// 30 Program Organization Units/FBs/AT_FUNKTIONEN/AT_ANTRIEB_STETIG/FB_AT_ANTRIEB_STETIG
FUNCTION_BLOCK FB_AT_ANTRIEB_STETIG EXTENDS FB_OBJ_ID_BASE
VAR_INPUT
	xRelease		:	BOOL;
	rRelease		:	REAL;
	xSafetyOk		:	BOOL;		
	xHand			:	BOOL;
	xRevision		:	BOOL;
	xAcknowledge	:	BOOL;
	rAcknowledge	:	REAL;
	xCosPhiOk		:	BOOL;
	xErrorAntrieb	:	BOOL;
END_VAR
VAR_OUTPUT
	(* Requests *)
	xHandPrio8	:	BOOL;
END_VAR
VAR
	(* BacNet Objects *)
	A_BO_1				:	WagoSysBACnet.FbBinaryOutput_large(-1);					// Schaltbefehl
	B_TL_1				:	WagoSysBACnet.FbTrendLog_large(-1);                     // Aufzeichnung Betrieb
	C_EE_1				:	WagoSysBACnet.FbEventEnrollment_large(-1);              // Instandhaltungsmeldung
	// Objekt D	wird nicht unterstützt KBOB 2017 AV KBOB 2021 PIV
	E_BV_2				:	WagoSysBACnet.FbBinaryValue_large(-1);                  // Handbetrieb
	F_BI_1				:	WagoSysBACnet.FbBinaryInput_large(-1);                  // Revisionsschalter
	G_AO_1				:	WagoSysBACnet.FbAnalogOutput_large(-1);                 // Sollwertvorgabe
	H_TL_2				:	WagoSysBACnet.FbTrendLog_large(-1);                     // Aufzeichnung Sollwert
	I_AI_1				:	WagoSysBACnet.FbAnalogInput_large(-1);                  // Istwert
	J_TL_3				:	WagoSysBACnet.FbTrendLog_large(-1);                     // Aufzeichnung Istwert
	K_BI_2				:	WagoSysBACnet.FbBinaryInput_large(-1);                  // Lauf Überwachung
	L_BV_3				:	WagoSysBACnet.FbBinaryValue_large(-1);					// Störung Antrieb
END_VAR
VAR CONSTANT
	usiAnzBacNetObj	:	USINT	:= 12;
END_VAR

(* Call Base FB*)
SUPER^();
(* Cyclic Action *)
IF xCreatet THEN
	(* DESCTIPTION FIX *)
	metCYCLIC_DESCRIPTION_FIX();
	(* Get Revision *)
	CASE GVL_BACNET.fbBacNetParameter.proKBOB_REV OF
		(* KBOB 2021 V2 *)
		enKBOB_REV.KBOB_REV2021_V2:
			metCYCLIC_KBOB_2021_V2();
		(* KBOB 2017 V1 *)
		enKBOB_REV.KBOB_REV2017_V1:
			metCYCLIC_KBOB_2017_V1();
		(* Default *)
		ELSE
			metCYCLIC_KBOB_2021_V2();
	END_CASE;	
END_IF;

METHOD metCYCLIC_KBOB_2017_V1
VAR_INPUT
END_VAR
(* A_BO_1 *)
	IF A_BO_1.IPriorityArray.aLevel[16].xValue <> xRelease THEN
		A_BO_1.IPriorityArray.SetPriority(16,xRelease,FALSE);	// Prio 16 Normal Command
	END_IF;
	IF NOT xSafetyOk THEN
		IF A_BO_1.IPriorityArray.aLevel[5].xNull THEN
			A_BO_1.IPriorityArray.SetPriority( 5,FALSE,FALSE);	// Prio  5 Device safety Off
		END_IF;
	ELSE
		IF NOT A_BO_1.IPriorityArray.aLevel[5].xNull THEN
			A_BO_1.IPriorityArray.SetPriority( 5,FALSE,TRUE);	// Prio  5 Device safety NULL
		END_IF;
	END_IF;	
	IF A_BO_1.xFeedbackValue <> xAcknowledge THEN
		A_BO_1.xFeedbackValue := xAcknowledge;
	END_IF;

	(* E_BV_2 *)
	IF E_BV_2.IPriorityArray.aLevel[16].xValue <> (xHand OR xRevision) THEN
		E_BV_2.IPriorityArray.SetPriority(16,xHand OR xRevision,FALSE);
	END_IF;
	(* F_BI_1 *)
	F_BI_1.xIN := xRevision;
	(* G_AO_1 *)
	IF G_AO_1.IPriorityArray.aLevel[5].rValue <> rRelease THEN
		G_AO_1.IPriorityArray.SetPriority(5,rRelease,FALSE);
	END_IF;
	(* I_AI_1 *)
	I_AI_1.rIN := rAcknowledge;
	(* K_BI_2 *)
	K_BI_2.xIN := xCosPhiOk;
	(* L_BV_3 *)
	L_BV_3.xPresentValue := xErrorAntrieb;
	
	(* Request Hand Prio 8 *)
	xHandPrio8 := NOT A_BO_1.IPriorityArray.aLevel[8].xNull AND A_BO_1.IPriorityArray.aLevel[8].xValue;
END_METHOD

METHOD metCYCLIC_KBOB_2021_V2
VAR_INPUT
END_VAR
(* A_BO_1 *)
	IF A_BO_1.IPriorityArray.aLevel[16].xValue <> xRelease THEN
		A_BO_1.IPriorityArray.SetPriority(16,xRelease,FALSE);	// Prio 16 Normal Command
	END_IF;
	IF NOT xSafetyOk THEN
		IF A_BO_1.IPriorityArray.aLevel[5].xNull THEN
			A_BO_1.IPriorityArray.SetPriority( 5,FALSE,FALSE);	// Prio  5 Device safety Off
		END_IF;
	ELSE
		IF NOT A_BO_1.IPriorityArray.aLevel[5].xNull THEN
			A_BO_1.IPriorityArray.SetPriority( 5,FALSE,TRUE);	// Prio  5 Device safety NULL
		END_IF;
	END_IF;	
	IF A_BO_1.xFeedbackValue <> xAcknowledge THEN
		A_BO_1.xFeedbackValue := xAcknowledge;
	END_IF;

	(* E_BV_2 *)
	IF E_BV_2.IPriorityArray.aLevel[16].xValue <> (xHand OR xRevision) THEN
		E_BV_2.IPriorityArray.SetPriority(16,xHand OR xRevision,FALSE);
	END_IF;
	(* F_BI_1 *)
	F_BI_1.xIN := xRevision;
	(* G_AO_1 *)
	IF G_AO_1.IPriorityArray.aLevel[5].rValue <> rRelease THEN
		G_AO_1.IPriorityArray.SetPriority(5,rRelease,FALSE);
	END_IF;
	(* I_AI_1 *)
	I_AI_1.rIN := rAcknowledge;
	(* K_BI_2 *)
	K_BI_2.xIN := xCosPhiOk;
	(* L_BV_3 *)
	L_BV_3.xPresentValue := xErrorAntrieb;
	
	(* Request Hand Prio 8 *)
	xHandPrio8 := NOT A_BO_1.IPriorityArray.aLevel[8].xNull AND A_BO_1.IPriorityArray.aLevel[8].xValue;
END_METHOD

METHOD metCYCLIC_DESCRIPTION_FIX
VAR_INPUT
END_VAR
(* A_BO_1 *)
IF A_BO_1.xIsCreated THEN
	IF A_BO_1.sDescription <> A_BO_1._sDescription THEN
		A_BO_1.sDescription := A_BO_1._sDescription;
	END_IF;
END_IF;

(* B_TL_1 *)
IF B_TL_1.xIsCreated THEN
	IF B_TL_1.sDescription <> B_TL_1._sDescription THEN
		B_TL_1.sDescription := B_TL_1._sDescription;
	END_IF;
END_IF;

(* C_EE_1 *)
IF C_EE_1.xIsCreated THEN
	IF C_EE_1.sDescription <> C_EE_1._sDescription THEN
		C_EE_1.sDescription := C_EE_1._sDescription;
	END_IF;
END_IF;

(* D_ *)
// Not Avaiable

(* E_BV_2 *)
IF E_BV_2.xIsCreated THEN
	IF E_BV_2.sDescription <> E_BV_2._sDescription THEN
		E_BV_2.sDescription := E_BV_2._sDescription;
	END_IF;
END_IF;

(* F_BI_1 *)
IF F_BI_1.xIsCreated THEN
	IF F_BI_1.sDescription <> F_BI_1._sDescription THEN
		F_BI_1.sDescription := F_BI_1._sDescription;
	END_IF;
END_IF;

(* G_AO_1 *)
IF G_AO_1.xIsCreated THEN
	IF G_AO_1.sDescription <> G_AO_1._sDescription THEN
		G_AO_1.sDescription := G_AO_1._sDescription;
	END_IF;
END_IF;

(* H_TL_2 *)
IF H_TL_2.xIsCreated THEN
	IF H_TL_2.sDescription <> H_TL_2._sDescription THEN
		H_TL_2.sDescription := H_TL_2._sDescription;
	END_IF;
END_IF;

(* I_AI_1 *)
IF I_AI_1.xIsCreated THEN
	IF I_AI_1.sDescription <> I_AI_1._sDescription THEN
		I_AI_1.sDescription := I_AI_1._sDescription;
	END_IF;
END_IF;

(* J_TL_3 *)
IF J_TL_3.xIsCreated THEN
	IF J_TL_3.sDescription <> J_TL_3._sDescription THEN
		J_TL_3.sDescription := J_TL_3._sDescription;
	END_IF;
END_IF;

(* K_BI_2 *)
IF K_BI_2.xIsCreated THEN
	IF K_BI_2.sDescription <> K_BI_2._sDescription THEN
		K_BI_2.sDescription := K_BI_2._sDescription;
	END_IF;
END_IF;

(* L_BV_3 *)
IF L_BV_3.xIsCreated THEN
	IF L_BV_3.sDescription <> L_BV_3._sDescription THEN
		L_BV_3.sDescription := L_BV_3._sDescription;
	END_IF;
END_IF;
END_METHOD

(*FB_Exit muss explizit implementiert werden. Wenn es eine Implementierung gibt, dann wird 
die Methode aufgerufen, bevor die Steuerung den Code der Funktionsbaustein-Instanz entfernt
(impliziter Aufruf. Der Rückgabewert wird nicht ausgewertet.*)
METHOD FB_Exit : BOOL
VAR_INPUT
	(* TRUE: Die Exit-Methode wird aufgerufen, um die Instanz zu verlassen, die hinterher kopiert wird Online-Change).  *)
	bInCopyCode	: BOOL;
END_VAR
(* A_BO_1*)
IF A_BO_1.xIsCreated THEN
	A_BO_1.Delete();
END_IF;	
(* B_TL_1 *)
IF B_TL_1.xIsCreated THEN
	B_TL_1.Delete();
END_IF;	
(* C_EE_1 *)
IF C_EE_1.xIsCreated THEN
	C_EE_1.Delete();
END_IF;
(* E_BV_2 *)
IF E_BV_2.xIsCreated THEN
	E_BV_2.Delete();
END_IF;
(* F_BI_1 *)
IF F_BI_1.xIsCreated THEN
	F_BI_1.Delete();	
END_IF;
(* G_AO_1 *)
IF G_AO_1.xIsCreated THEN
	G_AO_1.Delete();
END_IF;
(* H_TL_2 *)
IF H_TL_2.xIsCreated THEN
	H_TL_2.Delete();
END_IF;
(* I_AI_1 *)
IF I_AI_1.xIsCreated THEN
	I_AI_1.Delete();
END_IF;
(* J_TL_3 *)
IF J_TL_3.xIsCreated THEN
	J_TL_3.Delete();
END_IF;
(* K_BI_2 *)
IF K_BI_2.xIsCreated THEN
	K_BI_2.Delete();
END_IF;
(* L_BV_3 *)
IF L_BV_3.xIsCreated THEN
	L_BV_3.Delete();
END_IF;
END_METHOD

METHOD metDELETE : BOOL
VAR_INPUT
END_VAR
VAR
	oStatus		:	WagoSysErrorBase.FbResult;
END_VAR
(* A_BO_1*)
IF A_BO_1.xIsCreated THEN
	A_BO_1.Delete(oStatus=>oStatus);
END_IF;	
(* B_TL_1 *)
IF B_TL_1.xIsCreated THEN
	IF GVL_BACNET.fbBacNetParameter.proDestroyBacNetOverrideXmlNode THEN
		fcXMLDeleteOverrideNode(fcBacNetIdToIdWitType(B_TL_1.IObjectIdentifier.diInstance,B_TL_1.IObjectIdentifier.eObjectType));
	END_IF;
	B_TL_1.Delete(oStatus=>oStatus);
END_IF;	
(* C_EE_1 *)
IF C_EE_1.xIsCreated THEN
	C_EE_1.Delete(oStatus=>oStatus);
END_IF;
(* E_BV_2 *)
IF E_BV_2.xIsCreated THEN
	E_BV_2.Delete(oStatus=>oStatus);
END_IF;
(* F_BI_1 *)
IF F_BI_1.xIsCreated THEN
	F_BI_1.Delete(oStatus=>oStatus);	
END_IF;
(* G_AO_1 *)
IF G_AO_1.xIsCreated THEN
	G_AO_1.Delete(oStatus=>oStatus);
END_IF;
(* H_TL_2 *)
IF H_TL_2.xIsCreated THEN
	IF GVL_BACNET.fbBacNetParameter.proDestroyBacNetOverrideXmlNode THEN
		fcXMLDeleteOverrideNode(fcBacNetIdToIdWitType(H_TL_2.IObjectIdentifier.diInstance,H_TL_2.IObjectIdentifier.eObjectType));
	END_IF;
	H_TL_2.Delete(oStatus=>oStatus);
END_IF;
(* I_AI_1 *)
IF I_AI_1.xIsCreated THEN
	I_AI_1.Delete(oStatus=>oStatus);
END_IF;
(* J_TL_3 *)
IF J_TL_3.xIsCreated THEN
	IF GVL_BACNET.fbBacNetParameter.proDestroyBacNetOverrideXmlNode THEN
		fcXMLDeleteOverrideNode(fcBacNetIdToIdWitType(J_TL_3.IObjectIdentifier.diInstance,J_TL_3.IObjectIdentifier.eObjectType));
	END_IF;
	J_TL_3.Delete(oStatus=>oStatus);
END_IF;
(* K_BI_2 *)
IF K_BI_2.xIsCreated THEN
	K_BI_2.Delete(oStatus=>oStatus);
END_IF;
(* L_BV_3 *)
IF L_BV_3.xIsCreated THEN
	L_BV_3.Delete(oStatus=>oStatus);
END_IF;
(* Delete Struct View *)
IF GVL_BACNET.fbBacNetParameter.proDestroyBacNetOverrideXmlNode THEN
	fcXMLDeleteOverrideNode(fcBacNetIdToIdWitType(TO_DINT(CONCAT(TO_STRING(OBJ_ID_BASE),'1')),WagoTypesBacNet.eBACnetObjectType.BACnet_structured_view));
	fcXMLDeleteStructuredViewFromDevice(fcBacNetIdToIdWitType(TO_DINT(CONCAT(TO_STRING(OBJ_ID_BASE),'1')),WagoTypesBacNet.eBACnetObjectType.BACnet_structured_view));
END_IF;
metDELETE := 	A_BO_1.xIsCreated OR 
				B_TL_1.xIsCreated OR
				C_EE_1.xIsCreated OR				
				E_BV_2.xIsCreated OR
				F_BI_1.xIsCreated OR
				G_AO_1.xIsCreated OR
				I_AI_1.xIsCreated OR
				K_BI_2.xIsCreated OR
				L_BV_3.xIsCreated;
(* Reset Create Case *)
usiCreateCase := 1;
END_METHOD

METHOD metCREATE_KBOB_2017_V1 : BOOL;
VAR_INPUT
END_VAR
VAR
	oStatus		:	WagoSysErrorBase.FbResult;
	usiErrors	:	USINT;
END_VAR
(* Resett *)
usiErrors := 0;	

(* Create Objeccts *)
CASE usiCreateCase OF
	1:	
		usiErrors := usiErrors + TO_USINT(NOT metCreate_A_BO_1());
	2:
		usiErrors := usiErrors + TO_USINT(NOT metCreate_B_TL_1());
	3:	
		usiErrors := usiErrors + TO_USINT(NOT metCreate_C_EE_1());
	4:	
		;// Objekt D aus KBOB 2017 nicht realisierbar aufgrund fehlender Setpoint reference
	5:
		usiErrors := usiErrors + TO_USINT(NOT metCreate_E_BV_2());
	6:	
		usiErrors := usiErrors + TO_USINT(NOT metCreate_F_BI_1());
	7:
		usiErrors := usiErrors + TO_USINT(NOT metCreate_G_AO_1());
	8:	
		usiErrors := usiErrors + TO_USINT(NOT metCreate_H_TL_2());
	9:
		usiErrors := usiErrors + TO_USINT(NOT metCreate_I_AI_1());
	10:
		usiErrors := usiErrors + TO_USINT(NOT metCreate_J_TL_3());
	11:	
		usiErrors := usiErrors + TO_USINT(NOT metCreate_K_BI_2());
	12:
		usiErrors := usiErrors + TO_USINT(NOT metCreate_L_BV_3());
	0: 
		usiCreateCase := 1;
ELSE
	usiCreateCase := 0;
END_CASE;

(* STRUCT VIEW *)
metCREATE_STRUCTVIEW_KBOB_2017_V1();

(* OK = 0*)
metCREATE_KBOB_2017_V1 := NOT TO_BOOL(usiErrors);
END_METHOD

METHOD metCREATE_STRUCTVIEW_KBOB_2017_V1 : BOOL
VAR_INPUT
END_VAR
CASE usiCreateCase OF
	1:
		fcXMLStructuredView(THIS^,A_BO_1.IObjectIdentifier);
	2:
		fcXMLStructuredView(THIS^,B_TL_1.IObjectIdentifier);
	3:
		fcXMLStructuredView(THIS^,C_EE_1.IObjectIdentifier);
	4:
		;// Reserve für D
	5:
		fcXMLStructuredView(THIS^,E_BV_2.IObjectIdentifier);
	6:
		fcXMLStructuredView(THIS^,F_BI_1.IObjectIdentifier);
	7:
		fcXMLStructuredView(THIS^,G_AO_1.IObjectIdentifier);
	8:
		fcXMLStructuredView(THIS^,H_TL_2.IObjectIdentifier);
	9:
		fcXMLStructuredView(THIS^,I_AI_1.IObjectIdentifier);
	10:
		fcXMLStructuredView(THIS^,J_TL_3.IObjectIdentifier);
	11:
		fcXMLStructuredView(THIS^,K_BI_2.IObjectIdentifier);
	12:
		fcXMLStructuredView(THIS^,L_BV_3.IObjectIdentifier);
		fcXMLAddStructuredViewToDevice(THIS^);	
	0: 
		usiCreateCase := 1;
ELSE
	usiCreateCase := 0;
END_CASE
END_METHOD

METHOD metCREATE_STRUCTVIEW_KBOB_2021_V2 : BOOL
VAR_INPUT
END_VAR
CASE usiCreateCase OF
	1:
		fcXMLStructuredView(THIS^,A_BO_1.IObjectIdentifier);
	2:
		fcXMLStructuredView(THIS^,B_TL_1.IObjectIdentifier);
	3:
		fcXMLStructuredView(THIS^,C_EE_1.IObjectIdentifier);
	4:
		;// Reserve für D
	5:
		fcXMLStructuredView(THIS^,E_BV_2.IObjectIdentifier);
	6:
		fcXMLStructuredView(THIS^,F_BI_1.IObjectIdentifier);
	7:
		fcXMLStructuredView(THIS^,G_AO_1.IObjectIdentifier);
	8:
		fcXMLStructuredView(THIS^,H_TL_2.IObjectIdentifier);
	9:
		fcXMLStructuredView(THIS^,I_AI_1.IObjectIdentifier);
	10:
		fcXMLStructuredView(THIS^,J_TL_3.IObjectIdentifier);
	11:
		fcXMLStructuredView(THIS^,K_BI_2.IObjectIdentifier);
	12:
		fcXMLStructuredView(THIS^,L_BV_3.IObjectIdentifier);
		fcXMLAddStructuredViewToDevice(THIS^);	
	0: 
		usiCreateCase := 1;
ELSE
	usiCreateCase := 0;
END_CASE
END_METHOD

METHOD metCREATE_KBOB_2021_V2 : BOOL;
VAR_INPUT
END_VAR
VAR
	oStatus		:	WagoSysErrorBase.FbResult;
	usiErrors	:	USINT;
END_VAR
(* Resett *)
usiErrors := 0;	

(* Create Objeccts *)
CASE usiCreateCase OF
	1:	
		usiErrors := usiErrors + TO_USINT(NOT metCreate_A_BO_1());
	2:
		usiErrors := usiErrors + TO_USINT(NOT metCreate_B_TL_1());
	3:	
		usiErrors := usiErrors + TO_USINT(NOT metCreate_C_EE_1());
	4:	
		;// Objekt D aus KBOB 2017 nicht realisierbar aufgrund fehlender Setpoint reference
	5:
		usiErrors := usiErrors + TO_USINT(NOT metCreate_E_BV_2());
	6:	
		usiErrors := usiErrors + TO_USINT(NOT metCreate_F_BI_1());
	7:
		usiErrors := usiErrors + TO_USINT(NOT metCreate_G_AO_1());
	8:	
		usiErrors := usiErrors + TO_USINT(NOT metCreate_H_TL_2());
	9:
		usiErrors := usiErrors + TO_USINT(NOT metCreate_I_AI_1());
	10:
		usiErrors := usiErrors + TO_USINT(NOT metCreate_J_TL_3());
	11:	
		usiErrors := usiErrors + TO_USINT(NOT metCreate_K_BI_2());
	12:
		usiErrors := usiErrors + TO_USINT(NOT metCreate_L_BV_3());
	0: 
		usiCreateCase := 1;
ELSE
	usiCreateCase := 0;
END_CASE;

(* STRUCT VIEW *)
metCREATE_STRUCTVIEW_KBOB_2021_V2();

(* OK = 0*)
metCREATE_KBOB_2021_V2 := NOT TO_BOOL(usiErrors);
END_METHOD

METHOD metCREATE : BOOL;
VAR_INPUT
END_VAR
VAR
	oStatus		:	WagoSysErrorBase.FbResult;
	usiErrors	:	USINT;
END_VAR
(* Get Revision *)
CASE GVL_BACNET.fbBacNetParameter.proKBOB_REV OF
	(* KBOB 2021 V2 *)
	enKBOB_REV.KBOB_REV2021_V2:
		usiErrors := usiErrors + TO_USINT(NOT metCREATE_KBOB_2021_V2());
	(* KBOB 2017 V1 *)
	enKBOB_REV.KBOB_REV2017_V1:
		usiErrors := usiErrors + TO_USINT(NOT metCREATE_KBOB_2017_V1());
	(* Default *)
	ELSE
		usiErrors := usiErrors + TO_USINT(NOT metCREATE_KBOB_2021_V2());
END_CASE;

(* OK = 0*)
xErrorCreate := TO_BOOL(usiErrors);
metCREATE := NOT TO_BOOL(usiErrors) AND usiCreateCase = usiAnzBacNetObj;
END_METHOD

METHOD metCreate_F_BI_1 : BOOL
(* F_BI_1*)
IF NOT F_BI_1.xIsCreated THEN
	(* Ziel						UTF8->ASCII						OBJ_NAME_BASE			BacNet Text		Textlistname									BacNet Funktion																BacNet Textlist type												TextId		*)
	F_BI_1._sObjectName		:=	fcUtfToAscii(Standard.CONCAT(	OBJ_NAME_BASE		,	fcGetBcText(	GVL_BACNET.fbBacNetParameter.metGetTextListName(enTypeOfBacNetFunktionIn := enTypeOfBacNetFunktion.Type_AntriebStetig,		enTypeOfBacNetTextListIn := enTypeOfBacNetTextList.ENDING		),	'F_BI_1')));
	F_BI_1._sDescription	:= 	fcUtfToAscii(Standard.CONCAT(	OBJ_NAME_DESCRIPTION,	fcGetBcText(	GVL_BACNET.fbBacNetParameter.metGetTextListName(enTypeOfBacNetFunktionIn := enTypeOfBacNetFunktion.Type_AntriebStetig,		enTypeOfBacNetTextListIn := enTypeOfBacNetTextList.DESCRIPTION	),	'F_BI_1')));
	(* Create Id from Base Id and Object Nr (Last nummber of Name *)	
	F_BI_1.Create(diInstance := TO_DINT(Standard.CONCAT(TO_STRING(dwOBJ_ID_BASE),'1')));
	(* Check if Created *)
	IF F_BI_1.xIsCreated THEN
		(* Set Group *)
		F_BI_1.setPropertyGroup(WagoTypesBacNet.eBACnetPropertyIdentifier.PROP_PRESENT_VALUE						,WagoTypesBacNet.eBACnetPropertyUpdateGroup.GROUP_CYCLIC);
		F_BI_1.setPropertyGroup(WagoTypesBacNet.eBACnetPropertyIdentifier.PROP_PRIORITY_ARRAY						,WagoTypesBacNet.eBACnetPropertyUpdateGroup.GROUP_CYCLIC);
		F_BI_1.setPropertyGroup(WagoTypesBacNet.eBACnetPropertyIdentifier.PROP_ELAPSED_ACTIVE_TIME					,WagoTypesBacNet.eBACnetPropertyUpdateGroup.GROUP_CYCLIC);
		F_BI_1.setPropertyGroup(WagoTypesBacNet.eBACnetPropertyIdentifier.PROP_DESCRIPTION							,WagoTypesBacNet.eBACnetPropertyUpdateGroup.GROUP_CYCLIC);
		F_BI_1.setPropertyGroup(WagoTypesBacNet.eBACnetPropertyIdentifier.PROP_EVENT_MESSAGE_TEXTS_CONFIG			,WagoTypesBacNet.eBACnetPropertyUpdateGroup.GROUP_CYCLIC);
				
		(* Ziel												UTF8->ASCII		BacNet Text		Textlistname									BacNet Funktion																BacNet Textlist type												TextId		*)
		F_BI_1.IEventMessageTextsConfig.sToOffNormal	:=	fcUtfToAscii(	fcGetBcText(	GVL_BACNET.fbBacNetParameter.metGetTextListName(enTypeOfBacNetFunktionIn := enTypeOfBacNetFunktion.Type_AntriebStetig,		enTypeOfBacNetTextListIn := enTypeOfBacNetTextList.EVENTMESSAGE	),	'F_BI_1_ToOffNormal'	));		
		F_BI_1.IEventMessageTextsConfig.sToFault		:=	fcUtfToAscii(	fcGetBcText(	GVL_BACNET.fbBacNetParameter.metGetTextListName(enTypeOfBacNetFunktionIn := enTypeOfBacNetFunktion.Type_AntriebStetig,		enTypeOfBacNetTextListIn := enTypeOfBacNetTextList.EVENTMESSAGE	),	'F_BI_1_ToFault'		));		
		F_BI_1.IEventMessageTextsConfig.sToNormal		:=	fcUtfToAscii(	fcGetBcText(	GVL_BACNET.fbBacNetParameter.metGetTextListName(enTypeOfBacNetFunktionIn := enTypeOfBacNetFunktion.Type_AntriebStetig,		enTypeOfBacNetTextListIn := enTypeOfBacNetTextList.EVENTMESSAGE	),	'F_BI_1_ToNormal'		));		

		(* Ziel												UTF8->ASCII		BacNet Text		Textlistname									BacNet Funktion																BacNet Textlist type												TextId		*)	
		F_BI_1.sActiveText								:= 	fcUtfToAscii(	fcGetBcText(	GVL_BACNET.fbBacNetParameter.metGetTextListName(enTypeOfBacNetFunktionIn := enTypeOfBacNetFunktion.Type_AntriebStetig,		enTypeOfBacNetTextListIn := enTypeOfBacNetTextList.PRESENTVALUE	),	'F_BI_1_ST_ACTIVE'		));
		F_BI_1.sInactiveText							:= 	fcUtfToAscii(	fcGetBcText(	GVL_BACNET.fbBacNetParameter.metGetTextListName(enTypeOfBacNetFunktionIn := enTypeOfBacNetFunktion.Type_AntriebStetig,		enTypeOfBacNetTextListIn := enTypeOfBacNetTextList.PRESENTVALUE	),	'F_BI_1_ST_INACTIVE'	));	

		(* Ziel												Convert			BacNet Text		Textlistname									BacNet Funktion																BacNet Textlist type												TextId		*)	
		F_BI_1.udiNotificationClass						:= 	TO_UDINT	(	fcGetBcText(	GVL_BACNET.fbBacNetParameter.metGetTextListName(enTypeOfBacNetFunktionIn := enTypeOfBacNetFunktion.Type_AntriebStetig,		enTypeOfBacNetTextListIn := enTypeOfBacNetTextList.NC			),	'F_BI_1_NC'	));	
		F_BI_1.eNotifyType								:= 	WagoTypesBACnet.eBACnetNotifyType.NOTIFY_TYPE_EVENT;
		F_BI_1.xAlarmValue								:= 	TO_BOOL		(	fcGetBcText(	GVL_BACNET.fbBacNetParameter.metGetTextListName(enTypeOfBacNetFunktionIn := enTypeOfBacNetFunktion.Type_AntriebStetig,		enTypeOfBacNetTextListIn := enTypeOfBacNetTextList.NC			),	'F_BI_1_ALV'	));	
		
	ELSE
		F_BI_1.Delete();
	END_IF;
	(* Get Status *)
	metCreate_F_BI_1 := F_BI_1.xIsCreated;	
END_IF;
END_METHOD

METHOD metCreate_G_AO_1 : BOOL
(* G_AO_1*)
IF NOT G_AO_1.xIsCreated THEN
	(* Ziel						UTF8->ASCII						OBJ_NAME_BASE			BacNet Text		Textlistname									BacNet Funktion																BacNet Textlist type												TextId		*)
	G_AO_1._sObjectName		:=	fcUtfToAscii(Standard.CONCAT(	OBJ_NAME_BASE		,	fcGetBcText(	GVL_BACNET.fbBacNetParameter.metGetTextListName(enTypeOfBacNetFunktionIn := enTypeOfBacNetFunktion.Type_AntriebStetig,		enTypeOfBacNetTextListIn := enTypeOfBacNetTextList.ENDING		),	'G_AO_1')));
	G_AO_1._sDescription	:= 	fcUtfToAscii(Standard.CONCAT(	OBJ_NAME_DESCRIPTION,	fcGetBcText(	GVL_BACNET.fbBacNetParameter.metGetTextListName(enTypeOfBacNetFunktionIn := enTypeOfBacNetFunktion.Type_AntriebStetig,		enTypeOfBacNetTextListIn := enTypeOfBacNetTextList.DESCRIPTION	),	'G_AO_1')));
	(* Create Id from Base Id and Object Nr (Last nummber of Name *)	
	G_AO_1.Create(diInstance := TO_DINT(Standard.CONCAT(TO_STRING(dwOBJ_ID_BASE),'1')));
	(* Check if Created *)
	IF G_AO_1.xIsCreated THEN
		(* Set Group *)
		G_AO_1.setPropertyGroup(WagoTypesBacNet.eBACnetPropertyIdentifier.PROP_PRESENT_VALUE						,WagoTypesBacNet.eBACnetPropertyUpdateGroup.GROUP_CYCLIC);
		G_AO_1.setPropertyGroup(WagoTypesBacNet.eBACnetPropertyIdentifier.PROP_PRIORITY_ARRAY						,WagoTypesBacNet.eBACnetPropertyUpdateGroup.GROUP_CYCLIC);
		G_AO_1.setPropertyGroup(WagoTypesBacNet.eBACnetPropertyIdentifier.PROP_ELAPSED_ACTIVE_TIME					,WagoTypesBacNet.eBACnetPropertyUpdateGroup.GROUP_CYCLIC);
		G_AO_1.setPropertyGroup(WagoTypesBacNet.eBACnetPropertyIdentifier.PROP_DESCRIPTION							,WagoTypesBacNet.eBACnetPropertyUpdateGroup.GROUP_CYCLIC);
		G_AO_1.setPropertyGroup(WagoTypesBacNet.eBACnetPropertyIdentifier.PROP_EVENT_MESSAGE_TEXTS_CONFIG			,WagoTypesBacNet.eBACnetPropertyUpdateGroup.GROUP_CYCLIC);
				
		(* Ziel												UTF8->ASCII		BacNet Text		Textlistname									BacNet Funktion																BacNet Textlist type												TextId		*)
		G_AO_1.IEventMessageTextsConfig.sToOffNormal	:=	fcUtfToAscii(	fcGetBcText(	GVL_BACNET.fbBacNetParameter.metGetTextListName(enTypeOfBacNetFunktionIn := enTypeOfBacNetFunktion.Type_AntriebStetig,		enTypeOfBacNetTextListIn := enTypeOfBacNetTextList.EVENTMESSAGE	),	'G_AO_1_ToOffNormal'	));		
		G_AO_1.IEventMessageTextsConfig.sToFault		:=	fcUtfToAscii(	fcGetBcText(	GVL_BACNET.fbBacNetParameter.metGetTextListName(enTypeOfBacNetFunktionIn := enTypeOfBacNetFunktion.Type_AntriebStetig,		enTypeOfBacNetTextListIn := enTypeOfBacNetTextList.EVENTMESSAGE	),	'G_AO_1_ToFault'		));		
		G_AO_1.IEventMessageTextsConfig.sToNormal		:=	fcUtfToAscii(	fcGetBcText(	GVL_BACNET.fbBacNetParameter.metGetTextListName(enTypeOfBacNetFunktionIn := enTypeOfBacNetFunktion.Type_AntriebStetig,		enTypeOfBacNetTextListIn := enTypeOfBacNetTextList.EVENTMESSAGE	),	'G_AO_1_ToNormal'		));		

	ELSE
		G_AO_1.Delete();
	END_IF;
	(* Get Status *)
	metCreate_G_AO_1 := G_AO_1.xIsCreated;	
END_IF;
END_METHOD

METHOD metCreate_I_AI_1 : BOOL
(* I_AI_1*)
IF NOT I_AI_1.xIsCreated THEN
	(* Ziel						UTF8->ASCII						OBJ_NAME_BASE			BacNet Text		Textlistname									BacNet Funktion																BacNet Textlist type												TextId		*)
	I_AI_1._sObjectName		:=	fcUtfToAscii(Standard.CONCAT(	OBJ_NAME_BASE		,	fcGetBcText(	GVL_BACNET.fbBacNetParameter.metGetTextListName(enTypeOfBacNetFunktionIn := enTypeOfBacNetFunktion.Type_AntriebStetig,		enTypeOfBacNetTextListIn := enTypeOfBacNetTextList.ENDING		),	'I_AI_1')));
	I_AI_1._sDescription	:= 	fcUtfToAscii(Standard.CONCAT(	OBJ_NAME_DESCRIPTION,	fcGetBcText(	GVL_BACNET.fbBacNetParameter.metGetTextListName(enTypeOfBacNetFunktionIn := enTypeOfBacNetFunktion.Type_AntriebStetig,		enTypeOfBacNetTextListIn := enTypeOfBacNetTextList.DESCRIPTION	),	'I_AI_1')));
	(* Create Id from Base Id and Object Nr (Last nummber of Name *)	
	I_AI_1.Create(diInstance := TO_DINT(Standard.CONCAT(TO_STRING(dwOBJ_ID_BASE),'1')));
	(* Check if Created *)
	IF I_AI_1.xIsCreated THEN
		(* Set Group *)
		I_AI_1.setPropertyGroup(WagoTypesBacNet.eBACnetPropertyIdentifier.PROP_PRESENT_VALUE						,WagoTypesBacNet.eBACnetPropertyUpdateGroup.GROUP_CYCLIC);
		I_AI_1.setPropertyGroup(WagoTypesBacNet.eBACnetPropertyIdentifier.PROP_PRIORITY_ARRAY						,WagoTypesBacNet.eBACnetPropertyUpdateGroup.GROUP_CYCLIC);
		I_AI_1.setPropertyGroup(WagoTypesBacNet.eBACnetPropertyIdentifier.PROP_ELAPSED_ACTIVE_TIME					,WagoTypesBacNet.eBACnetPropertyUpdateGroup.GROUP_CYCLIC);
		I_AI_1.setPropertyGroup(WagoTypesBacNet.eBACnetPropertyIdentifier.PROP_DESCRIPTION							,WagoTypesBacNet.eBACnetPropertyUpdateGroup.GROUP_CYCLIC);
		I_AI_1.setPropertyGroup(WagoTypesBacNet.eBACnetPropertyIdentifier.PROP_EVENT_MESSAGE_TEXTS_CONFIG			,WagoTypesBacNet.eBACnetPropertyUpdateGroup.GROUP_CYCLIC);
		
		(* Ziel												UTF8->ASCII		BacNet Text		Textlistname									BacNet Funktion																BacNet Textlist type												TextId		*)
		I_AI_1.IEventMessageTextsConfig.sToOffNormal	:=	fcUtfToAscii(	fcGetBcText(	GVL_BACNET.fbBacNetParameter.metGetTextListName(enTypeOfBacNetFunktionIn := enTypeOfBacNetFunktion.Type_AntriebStetig,		enTypeOfBacNetTextListIn := enTypeOfBacNetTextList.EVENTMESSAGE	),	'I_AI_1_ToOffNormal'	));		
		I_AI_1.IEventMessageTextsConfig.sToFault		:=	fcUtfToAscii(	fcGetBcText(	GVL_BACNET.fbBacNetParameter.metGetTextListName(enTypeOfBacNetFunktionIn := enTypeOfBacNetFunktion.Type_AntriebStetig,		enTypeOfBacNetTextListIn := enTypeOfBacNetTextList.EVENTMESSAGE	),	'I_AI_1_ToFault'		));		
		I_AI_1.IEventMessageTextsConfig.sToNormal		:=	fcUtfToAscii(	fcGetBcText(	GVL_BACNET.fbBacNetParameter.metGetTextListName(enTypeOfBacNetFunktionIn := enTypeOfBacNetFunktion.Type_AntriebStetig,		enTypeOfBacNetTextListIn := enTypeOfBacNetTextList.EVENTMESSAGE	),	'I_AI_1_ToNormal'		));		

		(* Ziel												Convert			BacNet Text		Textlistname									BacNet Funktion																BacNet Textlist type												TextId		*)	
		I_AI_1.udiNotificationClass						:= 	TO_UDINT	(	fcGetBcText(	GVL_BACNET.fbBacNetParameter.metGetTextListName(enTypeOfBacNetFunktionIn := enTypeOfBacNetFunktion.Type_AntriebStetig,		enTypeOfBacNetTextListIn := enTypeOfBacNetTextList.NC			),	'I_AI_1_NC'	));	
		I_AI_1.eNotifyType								:= 	WagoTypesBACnet.eBACnetNotifyType.NOTIFY_TYPE_EVENT;
		
	ELSE
		I_AI_1.Delete();
	END_IF;
	(* Get Status *)
	metCreate_I_AI_1 := I_AI_1.xIsCreated;	
END_IF;
END_METHOD

METHOD metCreate_K_BI_2 : BOOL
(* K_BI_2*)
IF NOT K_BI_2.xIsCreated THEN
	(* Ziel						UTF8->ASCII						OBJ_NAME_BASE			BacNet Text		Textlistname									BacNet Funktion																BacNet Textlist type												TextId		*)
	K_BI_2._sObjectName		:=	fcUtfToAscii(Standard.CONCAT(	OBJ_NAME_BASE		,	fcGetBcText(	GVL_BACNET.fbBacNetParameter.metGetTextListName(enTypeOfBacNetFunktionIn := enTypeOfBacNetFunktion.Type_AntriebStetig,		enTypeOfBacNetTextListIn := enTypeOfBacNetTextList.ENDING		),	'K_BI_2')));
	K_BI_2._sDescription	:= 	fcUtfToAscii(Standard.CONCAT(	OBJ_NAME_DESCRIPTION,	fcGetBcText(	GVL_BACNET.fbBacNetParameter.metGetTextListName(enTypeOfBacNetFunktionIn := enTypeOfBacNetFunktion.Type_AntriebStetig,		enTypeOfBacNetTextListIn := enTypeOfBacNetTextList.DESCRIPTION	),	'K_BI_2')));
	(* Create Id from Base Id and Object Nr (Last nummber of Name *)	
	K_BI_2.Create(diInstance := TO_DINT(Standard.CONCAT(TO_STRING(dwOBJ_ID_BASE),'2')));
	(* Check if Created *)
	IF K_BI_2.xIsCreated THEN
		(* Set Group *)
		K_BI_2.setPropertyGroup(WagoTypesBacNet.eBACnetPropertyIdentifier.PROP_PRESENT_VALUE						,WagoTypesBacNet.eBACnetPropertyUpdateGroup.GROUP_CYCLIC);
		K_BI_2.setPropertyGroup(WagoTypesBacNet.eBACnetPropertyIdentifier.PROP_PRIORITY_ARRAY						,WagoTypesBacNet.eBACnetPropertyUpdateGroup.GROUP_CYCLIC);
		K_BI_2.setPropertyGroup(WagoTypesBacNet.eBACnetPropertyIdentifier.PROP_ELAPSED_ACTIVE_TIME					,WagoTypesBacNet.eBACnetPropertyUpdateGroup.GROUP_CYCLIC);
		K_BI_2.setPropertyGroup(WagoTypesBacNet.eBACnetPropertyIdentifier.PROP_DESCRIPTION							,WagoTypesBacNet.eBACnetPropertyUpdateGroup.GROUP_CYCLIC);
		K_BI_2.setPropertyGroup(WagoTypesBacNet.eBACnetPropertyIdentifier.PROP_EVENT_MESSAGE_TEXTS_CONFIG			,WagoTypesBacNet.eBACnetPropertyUpdateGroup.GROUP_CYCLIC);
		
		(* Ziel												UTF8->ASCII		BacNet Text		Textlistname									BacNet Funktion																BacNet Textlist type												TextId		*)
		K_BI_2.IEventMessageTextsConfig.sToOffNormal	:=	fcUtfToAscii(	fcGetBcText(	GVL_BACNET.fbBacNetParameter.metGetTextListName(enTypeOfBacNetFunktionIn := enTypeOfBacNetFunktion.Type_AntriebStetig,		enTypeOfBacNetTextListIn := enTypeOfBacNetTextList.EVENTMESSAGE	),	'K_BI_2_ToOffNormal'	));		
		K_BI_2.IEventMessageTextsConfig.sToFault		:=	fcUtfToAscii(	fcGetBcText(	GVL_BACNET.fbBacNetParameter.metGetTextListName(enTypeOfBacNetFunktionIn := enTypeOfBacNetFunktion.Type_AntriebStetig,		enTypeOfBacNetTextListIn := enTypeOfBacNetTextList.EVENTMESSAGE	),	'K_BI_2_ToFault'		));		
		K_BI_2.IEventMessageTextsConfig.sToNormal		:=	fcUtfToAscii(	fcGetBcText(	GVL_BACNET.fbBacNetParameter.metGetTextListName(enTypeOfBacNetFunktionIn := enTypeOfBacNetFunktion.Type_AntriebStetig,		enTypeOfBacNetTextListIn := enTypeOfBacNetTextList.EVENTMESSAGE	),	'K_BI_2_ToNormal'		));		

		(* Ziel												UTF8->ASCII		BacNet Text		Textlistname									BacNet Funktion																BacNet Textlist type												TextId		*)	
		K_BI_2.sActiveText								:= 	fcUtfToAscii(	fcGetBcText(	GVL_BACNET.fbBacNetParameter.metGetTextListName(enTypeOfBacNetFunktionIn := enTypeOfBacNetFunktion.Type_AntriebStetig,		enTypeOfBacNetTextListIn := enTypeOfBacNetTextList.PRESENTVALUE	),	'K_BI_2_ST_ACTIVE'		));
		K_BI_2.sInactiveText							:= 	fcUtfToAscii(	fcGetBcText(	GVL_BACNET.fbBacNetParameter.metGetTextListName(enTypeOfBacNetFunktionIn := enTypeOfBacNetFunktion.Type_AntriebStetig,		enTypeOfBacNetTextListIn := enTypeOfBacNetTextList.PRESENTVALUE	),	'K_BI_2_ST_INACTIVE'	));	

		(* Ziel												Convert			BacNet Text		Textlistname									BacNet Funktion																BacNet Textlist type												TextId		*)	
		K_BI_2.udiNotificationClass						:= 	TO_UDINT	(	fcGetBcText(	GVL_BACNET.fbBacNetParameter.metGetTextListName(enTypeOfBacNetFunktionIn := enTypeOfBacNetFunktion.Type_AntriebStetig,		enTypeOfBacNetTextListIn := enTypeOfBacNetTextList.NC			),	'K_BI_2_NC'	));	
		K_BI_2.eNotifyType								:= 	WagoTypesBACnet.eBACnetNotifyType.NOTIFY_TYPE_ALARM;
		K_BI_2.xAlarmValue								:= 	TO_BOOL		(	fcGetBcText(	GVL_BACNET.fbBacNetParameter.metGetTextListName(enTypeOfBacNetFunktionIn := enTypeOfBacNetFunktion.Type_AntriebStetig,		enTypeOfBacNetTextListIn := enTypeOfBacNetTextList.NC			),	'K_BI_2_ALV'	));	
		
	ELSE
		K_BI_2.Delete();
	END_IF;
	(* Get Status *)
	metCreate_K_BI_2 := K_BI_2.xIsCreated;	
END_IF;
END_METHOD

METHOD metCreate_L_BV_3 : BOOL
(* L_BV_3*)
IF NOT L_BV_3.xIsCreated THEN
	(* Ziel						UTF8->ASCII						OBJ_NAME_BASE			BacNet Text		Textlistname									BacNet Funktion																BacNet Textlist type												TextId		*)
	L_BV_3._sObjectName		:=	fcUtfToAscii(Standard.CONCAT(	OBJ_NAME_BASE		,	fcGetBcText(	GVL_BACNET.fbBacNetParameter.metGetTextListName(enTypeOfBacNetFunktionIn := enTypeOfBacNetFunktion.Type_AntriebStetig,		enTypeOfBacNetTextListIn := enTypeOfBacNetTextList.ENDING		),	'L_BV_3')));
	L_BV_3._sDescription	:= 	fcUtfToAscii(Standard.CONCAT(	OBJ_NAME_DESCRIPTION,	fcGetBcText(	GVL_BACNET.fbBacNetParameter.metGetTextListName(enTypeOfBacNetFunktionIn := enTypeOfBacNetFunktion.Type_AntriebStetig,		enTypeOfBacNetTextListIn := enTypeOfBacNetTextList.DESCRIPTION	),	'L_BV_3')));
	(* Create Id from Base Id and Object Nr (Last nummber of Name *)																
	L_BV_3.Create(diInstance := TO_DINT(Standard.CONCAT(TO_STRING(dwOBJ_ID_BASE),'3')));	
	(* Check if Created *)
	IF L_BV_3.xIsCreated THEN
		(* Set Group *)
		L_BV_3.setPropertyGroup(WagoTypesBacNet.eBACnetPropertyIdentifier.PROP_PRESENT_VALUE						,WagoTypesBacNet.eBACnetPropertyUpdateGroup.GROUP_CYCLIC);
		L_BV_3.setPropertyGroup(WagoTypesBacNet.eBACnetPropertyIdentifier.PROP_PRIORITY_ARRAY						,WagoTypesBacNet.eBACnetPropertyUpdateGroup.GROUP_CYCLIC);
		L_BV_3.setPropertyGroup(WagoTypesBacNet.eBACnetPropertyIdentifier.PROP_ELAPSED_ACTIVE_TIME					,WagoTypesBacNet.eBACnetPropertyUpdateGroup.GROUP_CYCLIC);
		L_BV_3.setPropertyGroup(WagoTypesBacNet.eBACnetPropertyIdentifier.PROP_DESCRIPTION							,WagoTypesBacNet.eBACnetPropertyUpdateGroup.GROUP_CYCLIC);
		L_BV_3.setPropertyGroup(WagoTypesBacNet.eBACnetPropertyIdentifier.PROP_EVENT_MESSAGE_TEXTS_CONFIG			,WagoTypesBacNet.eBACnetPropertyUpdateGroup.GROUP_CYCLIC);
				
		(* Ziel												UTF8->ASCII		BacNet Text		Textlistname									BacNet Funktion																BacNet Textlist type												TextId		*)
		L_BV_3.IEventMessageTextsConfig.sToOffNormal	:=	fcUtfToAscii(	fcGetBcText(	GVL_BACNET.fbBacNetParameter.metGetTextListName(enTypeOfBacNetFunktionIn := enTypeOfBacNetFunktion.Type_AntriebStetig,		enTypeOfBacNetTextListIn := enTypeOfBacNetTextList.EVENTMESSAGE	),	'L_BV_3_ToOffNormal'	));		
		L_BV_3.IEventMessageTextsConfig.sToFault		:=	fcUtfToAscii(	fcGetBcText(	GVL_BACNET.fbBacNetParameter.metGetTextListName(enTypeOfBacNetFunktionIn := enTypeOfBacNetFunktion.Type_AntriebStetig,		enTypeOfBacNetTextListIn := enTypeOfBacNetTextList.EVENTMESSAGE	),	'L_BV_3_ToFault'		));		
		L_BV_3.IEventMessageTextsConfig.sToNormal		:=	fcUtfToAscii(	fcGetBcText(	GVL_BACNET.fbBacNetParameter.metGetTextListName(enTypeOfBacNetFunktionIn := enTypeOfBacNetFunktion.Type_AntriebStetig,		enTypeOfBacNetTextListIn := enTypeOfBacNetTextList.EVENTMESSAGE	),	'L_BV_3_ToNormal'		));		

		(* Ziel												UTF8->ASCII		BacNet Text		Textlistname									BacNet Funktion																BacNet Textlist type												TextId		*)	
		L_BV_3.sActiveText								:= 	fcUtfToAscii(	fcGetBcText(	GVL_BACNET.fbBacNetParameter.metGetTextListName(enTypeOfBacNetFunktionIn := enTypeOfBacNetFunktion.Type_AntriebStetig,		enTypeOfBacNetTextListIn := enTypeOfBacNetTextList.PRESENTVALUE	),	'L_BV_3_ST_ACTIVE'		));
		L_BV_3.sInactiveText							:= 	fcUtfToAscii(	fcGetBcText(	GVL_BACNET.fbBacNetParameter.metGetTextListName(enTypeOfBacNetFunktionIn := enTypeOfBacNetFunktion.Type_AntriebStetig,		enTypeOfBacNetTextListIn := enTypeOfBacNetTextList.PRESENTVALUE	),	'L_BV_3_ST_INACTIVE'	));	

		(* Ziel												Convert			BacNet Text		Textlistname									BacNet Funktion																BacNet Textlist type												TextId		*)	
		L_BV_3.udiNotificationClass						:= 	TO_UDINT	(	fcGetBcText(	GVL_BACNET.fbBacNetParameter.metGetTextListName(enTypeOfBacNetFunktionIn := enTypeOfBacNetFunktion.Type_AntriebStetig,		enTypeOfBacNetTextListIn := enTypeOfBacNetTextList.NC			),	'L_BV_3_NC'	));	
		L_BV_3.eNotifyType								:= 	WagoTypesBACnet.eBACnetNotifyType.NOTIFY_TYPE_ALARM;
		L_BV_3.xAlarmValue								:= 	TO_BOOL		(	fcGetBcText(	GVL_BACNET.fbBacNetParameter.metGetTextListName(enTypeOfBacNetFunktionIn := enTypeOfBacNetFunktion.Type_AntriebStetig,		enTypeOfBacNetTextListIn := enTypeOfBacNetTextList.NC			),	'L_BV_3_ALV'	));	
		
	ELSE
		L_BV_3.Delete();
	END_IF;
	(* Get Status *)
	metCreate_L_BV_3 := L_BV_3.xIsCreated;	
END_IF;
END_METHOD

METHOD metCreate_H_TL_2 : BOOL
(* H_TL_2*)
IF NOT H_TL_2.xIsCreated THEN
	(* Ziel						UTF8->ASCII						OBJ_NAME_BASE			BacNet Text		Textlistname									BacNet Funktion																BacNet Textlist type												TextId		*)
	H_TL_2._sObjectName		:=	fcUtfToAscii(Standard.CONCAT(	OBJ_NAME_BASE		,	fcGetBcText(	GVL_BACNET.fbBacNetParameter.metGetTextListName(enTypeOfBacNetFunktionIn := enTypeOfBacNetFunktion.Type_AntriebStetig,		enTypeOfBacNetTextListIn := enTypeOfBacNetTextList.ENDING		),	'H_TL_2')));
	H_TL_2._sDescription	:= 	fcUtfToAscii(Standard.CONCAT(	OBJ_NAME_DESCRIPTION,	fcGetBcText(	GVL_BACNET.fbBacNetParameter.metGetTextListName(enTypeOfBacNetFunktionIn := enTypeOfBacNetFunktion.Type_AntriebStetig,		enTypeOfBacNetTextListIn := enTypeOfBacNetTextList.DESCRIPTION	),	'H_TL_2')));
	(* Create Id from Base Id and Object Nr (Last nummber of Name *)	
	H_TL_2.Create(diInstance := TO_DINT(Standard.CONCAT(TO_STRING(dwOBJ_ID_BASE),'2')));
	(* Check if Created *)
	IF H_TL_2.xIsCreated THEN
		(* Set Group *)
		H_TL_2.setPropertyGroup(WagoTypesBacNet.eBACnetPropertyIdentifier.PROP_PRESENT_VALUE						,WagoTypesBacNet.eBACnetPropertyUpdateGroup.GROUP_CYCLIC);
		H_TL_2.setPropertyGroup(WagoTypesBacNet.eBACnetPropertyIdentifier.PROP_PRIORITY_ARRAY						,WagoTypesBacNet.eBACnetPropertyUpdateGroup.GROUP_CYCLIC);
		H_TL_2.setPropertyGroup(WagoTypesBacNet.eBACnetPropertyIdentifier.PROP_ELAPSED_ACTIVE_TIME					,WagoTypesBacNet.eBACnetPropertyUpdateGroup.GROUP_CYCLIC);
		H_TL_2.setPropertyGroup(WagoTypesBacNet.eBACnetPropertyIdentifier.PROP_DESCRIPTION							,WagoTypesBacNet.eBACnetPropertyUpdateGroup.GROUP_CYCLIC);
		H_TL_2.setPropertyGroup(WagoTypesBacNet.eBACnetPropertyIdentifier.PROP_EVENT_MESSAGE_TEXTS_CONFIG			,WagoTypesBacNet.eBACnetPropertyUpdateGroup.GROUP_CYCLIC);
		
		(* Crate Override *)
		fcXMLTrendLogOverride(H_TL_2,G_AO_1.IObjectIdentifier,WagoTypesBacNet.eBACnetPropertyIdentifier.PROP_PRESENT_VALUE);
		
		(* Ziel												UTF8->ASCII		BacNet Text		Textlistname									BacNet Funktion																BacNet Textlist type												TextId		*)
		H_TL_2.IEventMessageTextsConfig.sToOffNormal	:=	fcUtfToAscii(	fcGetBcText(	GVL_BACNET.fbBacNetParameter.metGetTextListName(enTypeOfBacNetFunktionIn := enTypeOfBacNetFunktion.Type_AntriebStetig,		enTypeOfBacNetTextListIn := enTypeOfBacNetTextList.EVENTMESSAGE	),	'H_TL_2_ToOffNormal'	));		
		H_TL_2.IEventMessageTextsConfig.sToFault		:=	fcUtfToAscii(	fcGetBcText(	GVL_BACNET.fbBacNetParameter.metGetTextListName(enTypeOfBacNetFunktionIn := enTypeOfBacNetFunktion.Type_AntriebStetig,		enTypeOfBacNetTextListIn := enTypeOfBacNetTextList.EVENTMESSAGE	),	'H_TL_2_ToFault'		));		
		H_TL_2.IEventMessageTextsConfig.sToNormal		:=	fcUtfToAscii(	fcGetBcText(	GVL_BACNET.fbBacNetParameter.metGetTextListName(enTypeOfBacNetFunktionIn := enTypeOfBacNetFunktion.Type_AntriebStetig,		enTypeOfBacNetTextListIn := enTypeOfBacNetTextList.EVENTMESSAGE	),	'H_TL_2_ToNormal'		));		

		(* Ziel												Convert			BacNet Text		Textlistname									BacNet Funktion																BacNet Textlist type												TextId		*)	
		H_TL_2.udiNotificationClass						:= 	TO_UDINT	(	fcGetBcText(	GVL_BACNET.fbBacNetParameter.metGetTextListName(enTypeOfBacNetFunktionIn := enTypeOfBacNetFunktion.Type_AntriebStetig,		enTypeOfBacNetTextListIn := enTypeOfBacNetTextList.NC		),	'H_TL_2_NC'	));	
		H_TL_2.eNotifyType								:= 	WagoTypesBACnet.eBACnetNotifyType.NOTIFY_TYPE_EVENT;
			
		(* Logging Type *)
		H_TL_2.eLoggingType								:= WagoTypesBACnet.eBACnetLoggingType.LOGGING_TYPE_POLLED;
	
		(* Activate Logging *)
		H_TL_2.xEnable	:= TRUE;	
		
	ELSE
		H_TL_2.Delete();
	END_IF;
	(* Get Status *)
	metCreate_H_TL_2 := H_TL_2.xIsCreated;	
END_IF;
END_METHOD

METHOD metCreate_J_TL_3 : BOOL
(* J_TL_3*)
IF NOT J_TL_3.xIsCreated THEN
	(* Ziel						UTF8->ASCII						OBJ_NAME_BASE			BacNet Text		Textlistname									BacNet Funktion																BacNet Textlist type												TextId		*)
	J_TL_3._sObjectName		:=	fcUtfToAscii(Standard.CONCAT(	OBJ_NAME_BASE		,	fcGetBcText(	GVL_BACNET.fbBacNetParameter.metGetTextListName(enTypeOfBacNetFunktionIn := enTypeOfBacNetFunktion.Type_AntriebStetig,		enTypeOfBacNetTextListIn := enTypeOfBacNetTextList.ENDING		),	'J_TL_3')));
	J_TL_3._sDescription	:= 	fcUtfToAscii(Standard.CONCAT(	OBJ_NAME_DESCRIPTION,	fcGetBcText(	GVL_BACNET.fbBacNetParameter.metGetTextListName(enTypeOfBacNetFunktionIn := enTypeOfBacNetFunktion.Type_AntriebStetig,		enTypeOfBacNetTextListIn := enTypeOfBacNetTextList.DESCRIPTION	),	'J_TL_3')));
	(* Create Id from Base Id and Object Nr (Last nummber of Name *)	
	J_TL_3.Create(diInstance := TO_DINT(Standard.CONCAT(TO_STRING(dwOBJ_ID_BASE),'3')));
	(* Check if Created *)
	IF J_TL_3.xIsCreated THEN
		(* Set Group *)
		J_TL_3.setPropertyGroup(WagoTypesBacNet.eBACnetPropertyIdentifier.PROP_PRESENT_VALUE						,WagoTypesBacNet.eBACnetPropertyUpdateGroup.GROUP_CYCLIC);
		J_TL_3.setPropertyGroup(WagoTypesBacNet.eBACnetPropertyIdentifier.PROP_PRIORITY_ARRAY						,WagoTypesBacNet.eBACnetPropertyUpdateGroup.GROUP_CYCLIC);
		J_TL_3.setPropertyGroup(WagoTypesBacNet.eBACnetPropertyIdentifier.PROP_ELAPSED_ACTIVE_TIME					,WagoTypesBacNet.eBACnetPropertyUpdateGroup.GROUP_CYCLIC);
		J_TL_3.setPropertyGroup(WagoTypesBacNet.eBACnetPropertyIdentifier.PROP_DESCRIPTION							,WagoTypesBacNet.eBACnetPropertyUpdateGroup.GROUP_CYCLIC);
		J_TL_3.setPropertyGroup(WagoTypesBacNet.eBACnetPropertyIdentifier.PROP_EVENT_MESSAGE_TEXTS_CONFIG			,WagoTypesBacNet.eBACnetPropertyUpdateGroup.GROUP_CYCLIC);
		
		(* Crate Override *)
		fcXMLTrendLogOverride(J_TL_3,I_AI_1.IObjectIdentifier,WagoTypesBacNet.eBACnetPropertyIdentifier.PROP_PRESENT_VALUE);
		
		(* Ziel												UTF8->ASCII		BacNet Text		Textlistname									BacNet Funktion																BacNet Textlist type												TextId		*)
		J_TL_3.IEventMessageTextsConfig.sToOffNormal	:=	fcUtfToAscii(	fcGetBcText(	GVL_BACNET.fbBacNetParameter.metGetTextListName(enTypeOfBacNetFunktionIn := enTypeOfBacNetFunktion.Type_AntriebStetig,		enTypeOfBacNetTextListIn := enTypeOfBacNetTextList.EVENTMESSAGE	),	'J_TL_3_ToOffNormal'	));		
		J_TL_3.IEventMessageTextsConfig.sToFault		:=	fcUtfToAscii(	fcGetBcText(	GVL_BACNET.fbBacNetParameter.metGetTextListName(enTypeOfBacNetFunktionIn := enTypeOfBacNetFunktion.Type_AntriebStetig,		enTypeOfBacNetTextListIn := enTypeOfBacNetTextList.EVENTMESSAGE	),	'J_TL_3_ToFault'		));		
		J_TL_3.IEventMessageTextsConfig.sToNormal		:=	fcUtfToAscii(	fcGetBcText(	GVL_BACNET.fbBacNetParameter.metGetTextListName(enTypeOfBacNetFunktionIn := enTypeOfBacNetFunktion.Type_AntriebStetig,		enTypeOfBacNetTextListIn := enTypeOfBacNetTextList.EVENTMESSAGE	),	'J_TL_3_ToNormal'		));		

		(* Ziel												Convert			BacNet Text		Textlistname									BacNet Funktion																BacNet Textlist type												TextId		*)	
		J_TL_3.udiNotificationClass						:= 	TO_UDINT	(	fcGetBcText(	GVL_BACNET.fbBacNetParameter.metGetTextListName(enTypeOfBacNetFunktionIn := enTypeOfBacNetFunktion.Type_AntriebStetig,		enTypeOfBacNetTextListIn := enTypeOfBacNetTextList.NC		),	'J_TL_3_NC'	));	
		J_TL_3.eNotifyType								:= 	WagoTypesBACnet.eBACnetNotifyType.NOTIFY_TYPE_EVENT;

		(* Logging Type *)
		J_TL_3.eLoggingType								:= WagoTypesBACnet.eBACnetLoggingType.LOGGING_TYPE_POLLED;
		
		(* Activate Logging *)
		J_TL_3.xEnable	:= TRUE;
		
	ELSE
		J_TL_3.Delete();
	END_IF;
	(* Get Status *)
	metCreate_J_TL_3 := J_TL_3.xIsCreated;	
END_IF;
END_METHOD

METHOD metCreate_A_BO_1 : BOOL
(* A_BO_1*)
IF NOT A_BO_1.xIsCreated THEN
	(* Ziel						UTF8->ASCII						OBJ_NAME_BASE			BacNet Text		Textlistname									BacNet Funktion																BacNet Textlist type												TextId		*)
	A_BO_1._sObjectName		:=	fcUtfToAscii(Standard.CONCAT(	OBJ_NAME_BASE		,	fcGetBcText(	GVL_BACNET.fbBacNetParameter.metGetTextListName(enTypeOfBacNetFunktionIn := enTypeOfBacNetFunktion.Type_AntriebStetig,		enTypeOfBacNetTextListIn := enTypeOfBacNetTextList.ENDING		),	'A_BO_1')));
	A_BO_1._sDescription	:= 	fcUtfToAscii(Standard.CONCAT(	OBJ_NAME_DESCRIPTION,	fcGetBcText(	GVL_BACNET.fbBacNetParameter.metGetTextListName(enTypeOfBacNetFunktionIn := enTypeOfBacNetFunktion.Type_AntriebStetig,		enTypeOfBacNetTextListIn := enTypeOfBacNetTextList.DESCRIPTION	),	'A_BO_1')));
	(* Create Id from Base Id and Object Nr (Last nummber of Name *)	
	A_BO_1.Create(diInstance := TO_DINT(Standard.CONCAT(TO_STRING(dwOBJ_ID_BASE),'1')));
	(* Check if Created *)
	IF A_BO_1.xIsCreated THEN
		(* Set Group *)
		A_BO_1.setPropertyGroup(WagoTypesBacNet.eBACnetPropertyIdentifier.PROP_PRESENT_VALUE						,WagoTypesBacNet.eBACnetPropertyUpdateGroup.GROUP_CYCLIC);
		A_BO_1.setPropertyGroup(WagoTypesBacNet.eBACnetPropertyIdentifier.PROP_PRIORITY_ARRAY						,WagoTypesBacNet.eBACnetPropertyUpdateGroup.GROUP_CYCLIC);
		A_BO_1.setPropertyGroup(WagoTypesBacNet.eBACnetPropertyIdentifier.PROP_ELAPSED_ACTIVE_TIME					,WagoTypesBacNet.eBACnetPropertyUpdateGroup.GROUP_CYCLIC);
		A_BO_1.setPropertyGroup(WagoTypesBacNet.eBACnetPropertyIdentifier.PROP_DESCRIPTION							,WagoTypesBacNet.eBACnetPropertyUpdateGroup.GROUP_CYCLIC);
		A_BO_1.setPropertyGroup(WagoTypesBacNet.eBACnetPropertyIdentifier.PROP_EVENT_MESSAGE_TEXTS_CONFIG			,WagoTypesBacNet.eBACnetPropertyUpdateGroup.GROUP_CYCLIC);
			
		(* Ziel												UTF8->ASCII		BacNet Text		Textlistname									BacNet Funktion																BacNet Textlist type												TextId		*)
		A_BO_1.IEventMessageTextsConfig.sToOffNormal	:=	fcUtfToAscii(	fcGetBcText(	GVL_BACNET.fbBacNetParameter.metGetTextListName(enTypeOfBacNetFunktionIn := enTypeOfBacNetFunktion.Type_AntriebStetig,		enTypeOfBacNetTextListIn := enTypeOfBacNetTextList.EVENTMESSAGE	),	'A_BO_1_ToOffNormal'	));		
		A_BO_1.IEventMessageTextsConfig.sToFault		:=	fcUtfToAscii(	fcGetBcText(	GVL_BACNET.fbBacNetParameter.metGetTextListName(enTypeOfBacNetFunktionIn := enTypeOfBacNetFunktion.Type_AntriebStetig,		enTypeOfBacNetTextListIn := enTypeOfBacNetTextList.EVENTMESSAGE	),	'A_BO_1_ToFault'		));		
		A_BO_1.IEventMessageTextsConfig.sToNormal		:=	fcUtfToAscii(	fcGetBcText(	GVL_BACNET.fbBacNetParameter.metGetTextListName(enTypeOfBacNetFunktionIn := enTypeOfBacNetFunktion.Type_AntriebStetig,		enTypeOfBacNetTextListIn := enTypeOfBacNetTextList.EVENTMESSAGE	),	'A_BO_1_ToNormal'		));		

		(* Ziel												UTF8->ASCII		BacNet Text		Textlistname									BacNet Funktion																BacNet Textlist type												TextId		*)	
		A_BO_1.sActiveText								:= 	fcUtfToAscii(	fcGetBcText(	GVL_BACNET.fbBacNetParameter.metGetTextListName(enTypeOfBacNetFunktionIn := enTypeOfBacNetFunktion.Type_AntriebStetig,		enTypeOfBacNetTextListIn := enTypeOfBacNetTextList.PRESENTVALUE	),	'A_BO_1_ST_ACTIVE'		));
		A_BO_1.sInactiveText							:= 	fcUtfToAscii(	fcGetBcText(	GVL_BACNET.fbBacNetParameter.metGetTextListName(enTypeOfBacNetFunktionIn := enTypeOfBacNetFunktion.Type_AntriebStetig,		enTypeOfBacNetTextListIn := enTypeOfBacNetTextList.PRESENTVALUE	),	'A_BO_1_ST_INACTIVE'	));	

		(* Ziel												Convert			BacNet Text		Textlistname									BacNet Funktion																BacNet Textlist type												TextId		*)	
		A_BO_1.udiNotificationClass						:= 	TO_UDINT	(	fcGetBcText(	GVL_BACNET.fbBacNetParameter.metGetTextListName(enTypeOfBacNetFunktionIn := enTypeOfBacNetFunktion.Type_AntriebStetig,		enTypeOfBacNetTextListIn := enTypeOfBacNetTextList.NC			),	'A_BO_1_NC'	));	
		A_BO_1.eNotifyType								:= 	WagoTypesBACnet.eBACnetNotifyType.NOTIFY_TYPE_EVENT;
		
	ELSE
		A_BO_1.Delete();
	END_IF;
	(* Get Status *)
	metCreate_A_BO_1 := A_BO_1.xIsCreated;	
END_IF;
END_METHOD

METHOD metCreate_B_TL_1 : BOOL
VAR

END_VAR
(* B_TL_1*)
IF NOT B_TL_1.xIsCreated THEN
	(* Ziel						UTF8->ASCII						OBJ_NAME_BASE			BacNet Text		Textlistname									BacNet Funktion																BacNet Textlist type												TextId		*)
	B_TL_1._sObjectName		:=	fcUtfToAscii(Standard.CONCAT(	OBJ_NAME_BASE		,	fcGetBcText(	GVL_BACNET.fbBacNetParameter.metGetTextListName(enTypeOfBacNetFunktionIn := enTypeOfBacNetFunktion.Type_AntriebStetig,		enTypeOfBacNetTextListIn := enTypeOfBacNetTextList.ENDING		),	'B_TL_1')));
	B_TL_1._sDescription	:= 	fcUtfToAscii(Standard.CONCAT(	OBJ_NAME_DESCRIPTION,	fcGetBcText(	GVL_BACNET.fbBacNetParameter.metGetTextListName(enTypeOfBacNetFunktionIn := enTypeOfBacNetFunktion.Type_AntriebStetig,		enTypeOfBacNetTextListIn := enTypeOfBacNetTextList.DESCRIPTION	),	'B_TL_1')));
	(* Create Id from Base Id and Object Nr (Last nummber of Name *)	
	B_TL_1.Create(diInstance := TO_DINT(Standard.CONCAT(TO_STRING(dwOBJ_ID_BASE),'1')));
	(* Check if Created *)
	IF B_TL_1.xIsCreated THEN
		(* Set Group *)
		B_TL_1.setPropertyGroup(WagoTypesBacNet.eBACnetPropertyIdentifier.PROP_PRESENT_VALUE						,WagoTypesBacNet.eBACnetPropertyUpdateGroup.GROUP_CYCLIC);
		B_TL_1.setPropertyGroup(WagoTypesBacNet.eBACnetPropertyIdentifier.PROP_PRIORITY_ARRAY						,WagoTypesBacNet.eBACnetPropertyUpdateGroup.GROUP_CYCLIC);
		B_TL_1.setPropertyGroup(WagoTypesBacNet.eBACnetPropertyIdentifier.PROP_ELAPSED_ACTIVE_TIME					,WagoTypesBacNet.eBACnetPropertyUpdateGroup.GROUP_CYCLIC);
		B_TL_1.setPropertyGroup(WagoTypesBacNet.eBACnetPropertyIdentifier.PROP_DESCRIPTION							,WagoTypesBacNet.eBACnetPropertyUpdateGroup.GROUP_CYCLIC);
		B_TL_1.setPropertyGroup(WagoTypesBacNet.eBACnetPropertyIdentifier.PROP_EVENT_MESSAGE_TEXTS_CONFIG			,WagoTypesBacNet.eBACnetPropertyUpdateGroup.GROUP_CYCLIC);
		
		(* Crate Override *)
		fcXMLTrendLogOverride(B_TL_1,A_BO_1.IObjectIdentifier,WagoTypesBacNet.eBACnetPropertyIdentifier.PROP_FEEDBACK_VALUE);
		
		(* Ziel												UTF8->ASCII		BacNet Text		Textlistname									BacNet Funktion																BacNet Textlist type												TextId		*)
		B_TL_1.IEventMessageTextsConfig.sToOffNormal	:=	fcUtfToAscii(	fcGetBcText(	GVL_BACNET.fbBacNetParameter.metGetTextListName(enTypeOfBacNetFunktionIn := enTypeOfBacNetFunktion.Type_AntriebStetig,		enTypeOfBacNetTextListIn := enTypeOfBacNetTextList.EVENTMESSAGE	),	'B_TL_1_ToOffNormal'	));		
		B_TL_1.IEventMessageTextsConfig.sToFault		:=	fcUtfToAscii(	fcGetBcText(	GVL_BACNET.fbBacNetParameter.metGetTextListName(enTypeOfBacNetFunktionIn := enTypeOfBacNetFunktion.Type_AntriebStetig,		enTypeOfBacNetTextListIn := enTypeOfBacNetTextList.EVENTMESSAGE	),	'B_TL_1_ToFault'		));		
		B_TL_1.IEventMessageTextsConfig.sToNormal		:=	fcUtfToAscii(	fcGetBcText(	GVL_BACNET.fbBacNetParameter.metGetTextListName(enTypeOfBacNetFunktionIn := enTypeOfBacNetFunktion.Type_AntriebStetig,		enTypeOfBacNetTextListIn := enTypeOfBacNetTextList.EVENTMESSAGE	),	'B_TL_1_ToNormal'		));		

		(* Ziel												Convert			BacNet Text		Textlistname									BacNet Funktion																BacNet Textlist type												TextId		*)	
		B_TL_1.udiNotificationClass						:= 	TO_UDINT	(	fcGetBcText(	GVL_BACNET.fbBacNetParameter.metGetTextListName(enTypeOfBacNetFunktionIn := enTypeOfBacNetFunktion.Type_AntriebStetig,		enTypeOfBacNetTextListIn := enTypeOfBacNetTextList.NC		),	'B_TL_1_NC'	));	
		B_TL_1.eNotifyType								:= 	WagoTypesBACnet.eBACnetNotifyType.NOTIFY_TYPE_EVENT;
		
		(* Logging Type *)
		B_TL_1.eLoggingType								:= WagoTypesBACnet.eBACnetLoggingType.LOGGING_TYPE_POLLED;
		
		(* Activate Logging *)
		B_TL_1.xEnable	:= TRUE;	
								
	ELSE
		B_TL_1.Delete();
	END_IF;
	(* Get Status *)
	metCreate_B_TL_1 := B_TL_1.xIsCreated;	
END_IF;
END_METHOD

METHOD metCreate_C_EE_1 : BOOL
(* C_EE_1*)
IF NOT C_EE_1.xIsCreated THEN
	(* Ziel						UTF8->ASCII						OBJ_NAME_BASE			BacNet Text		Textlistname									BacNet Funktion																BacNet Textlist type												TextId		*)
	C_EE_1._sObjectName		:=	fcUtfToAscii(Standard.CONCAT(	OBJ_NAME_BASE		,	fcGetBcText(	GVL_BACNET.fbBacNetParameter.metGetTextListName(enTypeOfBacNetFunktionIn := enTypeOfBacNetFunktion.Type_AntriebStetig,		enTypeOfBacNetTextListIn := enTypeOfBacNetTextList.ENDING		),	'C_EE_1')));
	C_EE_1._sDescription	:= 	fcUtfToAscii(Standard.CONCAT(	OBJ_NAME_DESCRIPTION,	fcGetBcText(	GVL_BACNET.fbBacNetParameter.metGetTextListName(enTypeOfBacNetFunktionIn := enTypeOfBacNetFunktion.Type_AntriebStetig,		enTypeOfBacNetTextListIn := enTypeOfBacNetTextList.DESCRIPTION	),	'C_EE_1')));
	(* Create Id from Base Id and Object Nr (Last nummber of Name *)	
	C_EE_1.Create(diInstance := TO_DINT(Standard.CONCAT(TO_STRING(dwOBJ_ID_BASE),'1')));
	(* Check if Created *)
	IF C_EE_1.xIsCreated THEN
		(* Set Group *)
		C_EE_1.setPropertyGroup(WagoTypesBacNet.eBACnetPropertyIdentifier.PROP_PRESENT_VALUE						,WagoTypesBacNet.eBACnetPropertyUpdateGroup.GROUP_CYCLIC);
		C_EE_1.setPropertyGroup(WagoTypesBacNet.eBACnetPropertyIdentifier.PROP_PRIORITY_ARRAY						,WagoTypesBacNet.eBACnetPropertyUpdateGroup.GROUP_CYCLIC);
		C_EE_1.setPropertyGroup(WagoTypesBacNet.eBACnetPropertyIdentifier.PROP_ELAPSED_ACTIVE_TIME					,WagoTypesBacNet.eBACnetPropertyUpdateGroup.GROUP_CYCLIC);
		C_EE_1.setPropertyGroup(WagoTypesBacNet.eBACnetPropertyIdentifier.PROP_DESCRIPTION							,WagoTypesBacNet.eBACnetPropertyUpdateGroup.GROUP_CYCLIC);
		C_EE_1.setPropertyGroup(WagoTypesBacNet.eBACnetPropertyIdentifier.PROP_EVENT_MESSAGE_TEXTS_CONFIG			,WagoTypesBacNet.eBACnetPropertyUpdateGroup.GROUP_CYCLIC);
				
		(* Ziel												UTF8->ASCII		BacNet Text		Textlistname									BacNet Funktion																BacNet Textlist type												TextId		*)
		C_EE_1.IEventMessageTextsConfig.sToOffNormal	:=	fcUtfToAscii(	fcGetBcText(	GVL_BACNET.fbBacNetParameter.metGetTextListName(enTypeOfBacNetFunktionIn := enTypeOfBacNetFunktion.Type_AntriebStetig,		enTypeOfBacNetTextListIn := enTypeOfBacNetTextList.EVENTMESSAGE	),	'C_EE_1_ToOffNormal'	));		
		C_EE_1.IEventMessageTextsConfig.sToFault		:=	fcUtfToAscii(	fcGetBcText(	GVL_BACNET.fbBacNetParameter.metGetTextListName(enTypeOfBacNetFunktionIn := enTypeOfBacNetFunktion.Type_AntriebStetig,		enTypeOfBacNetTextListIn := enTypeOfBacNetTextList.EVENTMESSAGE	),	'C_EE_1_ToFault'		));		
		C_EE_1.IEventMessageTextsConfig.sToNormal		:=	fcUtfToAscii(	fcGetBcText(	GVL_BACNET.fbBacNetParameter.metGetTextListName(enTypeOfBacNetFunktionIn := enTypeOfBacNetFunktion.Type_AntriebStetig,		enTypeOfBacNetTextListIn := enTypeOfBacNetTextList.EVENTMESSAGE	),	'C_EE_1_ToNormal'		));		

		(* Ziel												Convert			BacNet Text		Textlistname									BacNet Funktion																BacNet Textlist type												TextId		*)	
		C_EE_1.udiNotificationClass						:= 	TO_UDINT	(	fcGetBcText(	GVL_BACNET.fbBacNetParameter.metGetTextListName(enTypeOfBacNetFunktionIn := enTypeOfBacNetFunktion.Type_AntriebStetig,		enTypeOfBacNetTextListIn := enTypeOfBacNetTextList.NC			),	'C_EE_1_NC'	));	
		C_EE_1.eNotifyType								:= 	WagoTypesBACnet.eBACnetNotifyType.NOTIFY_TYPE_EVENT;
		
	ELSE
		C_EE_1.Delete();
	END_IF;
	(* Get Status *)
	metCreate_C_EE_1 := C_EE_1.xIsCreated;	
END_IF;
END_METHOD

METHOD metCreate_E_BV_2 : BOOL
(* E_BV_2*)
IF NOT E_BV_2.xIsCreated THEN
	(* Ziel						UTF8->ASCII						OBJ_NAME_BASE			BacNet Text		Textlistname									BacNet Funktion																BacNet Textlist type												TextId		*)
	E_BV_2._sObjectName		:=	fcUtfToAscii(Standard.CONCAT(	OBJ_NAME_BASE		,	fcGetBcText(	GVL_BACNET.fbBacNetParameter.metGetTextListName(enTypeOfBacNetFunktionIn := enTypeOfBacNetFunktion.Type_AntriebStetig,		enTypeOfBacNetTextListIn := enTypeOfBacNetTextList.ENDING		),	'E_BV_2')));
	E_BV_2._sDescription	:= 	fcUtfToAscii(Standard.CONCAT(	OBJ_NAME_DESCRIPTION,	fcGetBcText(	GVL_BACNET.fbBacNetParameter.metGetTextListName(enTypeOfBacNetFunktionIn := enTypeOfBacNetFunktion.Type_AntriebStetig,		enTypeOfBacNetTextListIn := enTypeOfBacNetTextList.DESCRIPTION	),	'E_BV_2')));
	(* Create Id from Base Id and Object Nr (Last nummber of Name *)	
	E_BV_2.Create(diInstance := TO_DINT(Standard.CONCAT(TO_STRING(dwOBJ_ID_BASE),'2')));
	(* Check if Created *)
	IF E_BV_2.xIsCreated THEN
		(* Set Group *)
		E_BV_2.setPropertyGroup(WagoTypesBacNet.eBACnetPropertyIdentifier.PROP_PRESENT_VALUE						,WagoTypesBacNet.eBACnetPropertyUpdateGroup.GROUP_CYCLIC);
		E_BV_2.setPropertyGroup(WagoTypesBacNet.eBACnetPropertyIdentifier.PROP_PRIORITY_ARRAY						,WagoTypesBacNet.eBACnetPropertyUpdateGroup.GROUP_CYCLIC);
		E_BV_2.setPropertyGroup(WagoTypesBacNet.eBACnetPropertyIdentifier.PROP_ELAPSED_ACTIVE_TIME					,WagoTypesBacNet.eBACnetPropertyUpdateGroup.GROUP_CYCLIC);
		E_BV_2.setPropertyGroup(WagoTypesBacNet.eBACnetPropertyIdentifier.PROP_DESCRIPTION							,WagoTypesBacNet.eBACnetPropertyUpdateGroup.GROUP_CYCLIC);
		E_BV_2.setPropertyGroup(WagoTypesBacNet.eBACnetPropertyIdentifier.PROP_EVENT_MESSAGE_TEXTS_CONFIG			,WagoTypesBacNet.eBACnetPropertyUpdateGroup.GROUP_CYCLIC);
				
		(* Ziel												UTF8->ASCII		BacNet Text		Textlistname									BacNet Funktion																BacNet Textlist type												TextId		*)
		E_BV_2.IEventMessageTextsConfig.sToOffNormal	:=	fcUtfToAscii(	fcGetBcText(	GVL_BACNET.fbBacNetParameter.metGetTextListName(enTypeOfBacNetFunktionIn := enTypeOfBacNetFunktion.Type_AntriebStetig,		enTypeOfBacNetTextListIn := enTypeOfBacNetTextList.EVENTMESSAGE	),	'E_BV_2_ToOffNormal'	));		
		E_BV_2.IEventMessageTextsConfig.sToFault		:=	fcUtfToAscii(	fcGetBcText(	GVL_BACNET.fbBacNetParameter.metGetTextListName(enTypeOfBacNetFunktionIn := enTypeOfBacNetFunktion.Type_AntriebStetig,		enTypeOfBacNetTextListIn := enTypeOfBacNetTextList.EVENTMESSAGE	),	'E_BV_2_ToFault'		));		
		E_BV_2.IEventMessageTextsConfig.sToNormal		:=	fcUtfToAscii(	fcGetBcText(	GVL_BACNET.fbBacNetParameter.metGetTextListName(enTypeOfBacNetFunktionIn := enTypeOfBacNetFunktion.Type_AntriebStetig,		enTypeOfBacNetTextListIn := enTypeOfBacNetTextList.EVENTMESSAGE	),	'E_BV_2_ToNormal'		));		

		(* Ziel												UTF8->ASCII		BacNet Text		Textlistname									BacNet Funktion																BacNet Textlist type												TextId		*)	
		E_BV_2.sActiveText								:= 	fcUtfToAscii(	fcGetBcText(	GVL_BACNET.fbBacNetParameter.metGetTextListName(enTypeOfBacNetFunktionIn := enTypeOfBacNetFunktion.Type_AntriebStetig,		enTypeOfBacNetTextListIn := enTypeOfBacNetTextList.PRESENTVALUE	),	'E_BV_2_ST_ACTIVE'		));
		E_BV_2.sInactiveText							:= 	fcUtfToAscii(	fcGetBcText(	GVL_BACNET.fbBacNetParameter.metGetTextListName(enTypeOfBacNetFunktionIn := enTypeOfBacNetFunktion.Type_AntriebStetig,		enTypeOfBacNetTextListIn := enTypeOfBacNetTextList.PRESENTVALUE	),	'E_BV_2_ST_INACTIVE'	));	

		(* Ziel												Convert			BacNet Text		Textlistname									BacNet Funktion																BacNet Textlist type												TextId		*)	
		E_BV_2.udiNotificationClass						:= 	TO_UDINT	(	fcGetBcText(	GVL_BACNET.fbBacNetParameter.metGetTextListName(enTypeOfBacNetFunktionIn := enTypeOfBacNetFunktion.Type_AntriebStetig,		enTypeOfBacNetTextListIn := enTypeOfBacNetTextList.NC			),	'E_BV_2_NC'	));	
		E_BV_2.eNotifyType								:= 	WagoTypesBACnet.eBACnetNotifyType.NOTIFY_TYPE_EVENT;
		E_BV_2.xAlarmValue								:= 	TO_BOOL		(	fcGetBcText(	GVL_BACNET.fbBacNetParameter.metGetTextListName(enTypeOfBacNetFunktionIn := enTypeOfBacNetFunktion.Type_AntriebStetig,		enTypeOfBacNetTextListIn := enTypeOfBacNetTextList.NC			),	'E_BV_2_ALV'	));	
		
	ELSE
		E_BV_2.Delete();
	END_IF;
	(* Get Status *)
	metCreate_E_BV_2 := E_BV_2.xIsCreated;	
END_IF;
END_METHOD

END_FUNCTION_BLOCK

// 30 Program Organization Units/FBs/AT_FUNKTIONEN/AT_ANLAGENSCHALTER/FB_AT_ANLAGENSCHALTER
FUNCTION_BLOCK FB_AT_ANLAGENSCHALTER EXTENDS FB_OBJ_ID_BASE
VAR_INPUT
	xAutoIn			:	BOOL;
	xHandOffIn		:	BOOL;
	xHandOnIn		:	BOOL;
END_VAR
VAR_OUTPUT
	xAutoOut		:	BOOL;
	xHandOut		:	BOOL;
	xOffOut			:	BOOL;
	xOnOut			:	BOOL;													
END_VAR
VAR
	(* BacNet Objects *)
	A_MV_1			:	WagoSysBACnet.FbMultistateValue_large(-1);				// Betriebswahl					
	B_MI_1			:	WagoSysBACnet.FbMultistateInput_large(-1);              // Betriebswahl Lokal
	C_BV_1			:	WagoSysBACnet.FbBinaryValue_large(-1);              	// Handbetrieb / nicht Auto
	D_SC_1			:	WagoSysBACnet.FbSchedule_large(-1);                  	// Zeitschaltuhr	
END_VAR
VAR CONSTANT
	usiAnzBacNetObj	:	USINT	:= 4;
END_VAR

(* Call Base FB*)
SUPER^();
(* Cyclic Action *)
IF xCreatet THEN
	(* DESCTIPTION FIX *)
	metCYCLIC_DESCRIPTION_FIX();	
	(* Get Revision *)
	CASE GVL_BACNET.fbBacNetParameter.proKBOB_REV OF
		(* KBOB 2021 V2 *)
		enKBOB_REV.KBOB_REV2021_V2:
			metCYCLIC_KBOB_2021_V2();
		(* KBOB 2017 V1 *)
		enKBOB_REV.KBOB_REV2017_V1:
			metCYCLIC_KBOB_2017_V1();
		(* Default *)
		ELSE
			metCYCLIC_KBOB_2021_V2();
	END_CASE;	
END_IF;

(*FB_Exit muss explizit implementiert werden. Wenn es eine Implementierung gibt, dann wird 
die Methode aufgerufen, bevor die Steuerung den Code der Funktionsbaustein-Instanz entfernt
(impliziter Aufruf. Der Rückgabewert wird nicht ausgewertet.*)
METHOD FB_Exit : BOOL
VAR_INPUT
	(* TRUE: Die Exit-Methode wird aufgerufen, um die Instanz zu verlassen, die hinterher kopiert wird Online-Change).  *)
	bInCopyCode	: BOOL;
END_VAR
(* A_MV_1*)
IF A_MV_1.xIsCreated THEN
	A_MV_1.Delete();
END_IF;	
(* B_MI_1 *)
IF B_MI_1.xIsCreated THEN
		B_MI_1.Delete();
END_IF;	
(* C_BV_1 *)
IF C_BV_1.xIsCreated THEN
	C_BV_1.Delete();
END_IF;
(* D_SC_1 *)
IF D_SC_1.xIsCreated THEN
	D_SC_1.Delete();	
END_IF;
END_METHOD

METHOD metCREATE : BOOL;
VAR_INPUT
END_VAR
VAR
	usiErrors	:	USINT;
END_VAR
(* Get Revision *)
CASE GVL_BACNET.fbBacNetParameter.proKBOB_REV OF
	(* KBOB 2021 V2 *)
	enKBOB_REV.KBOB_REV2021_V2:
		usiErrors := usiErrors + TO_USINT(NOT metCREATE_KBOB_2021_V2());
	(* KBOB 2017 V1 *)
	enKBOB_REV.KBOB_REV2017_V1:
		usiErrors := usiErrors + TO_USINT(NOT metCREATE_KBOB_2017_V1());
	(* Default *)
	ELSE
		usiErrors := usiErrors + TO_USINT(NOT metCREATE_KBOB_2021_V2());
END_CASE;

(* OK = 0*)
xErrorCreate := TO_BOOL(usiErrors);
metCREATE := NOT TO_BOOL(usiErrors) AND usiCreateCase = usiAnzBacNetObj;
END_METHOD

METHOD metCreate_A_MV_1 : BOOL
(* A_MV_1*)
IF NOT A_MV_1.xIsCreated THEN
	(* Ziel						UTF8->ASCII						OBJ_NAME_BASE			BacNet Text		Textlistname									BacNet Funktion																BacNet Textlist type												TextId		*)
	A_MV_1._sObjectName		:=	fcUtfToAscii(Standard.CONCAT(	OBJ_NAME_BASE		,	fcGetBcText(	GVL_BACNET.fbBacNetParameter.metGetTextListName(enTypeOfBacNetFunktionIn := enTypeOfBacNetFunktion.Type_Anlagenschalter,	enTypeOfBacNetTextListIn := enTypeOfBacNetTextList.ENDING		),	'A_MV_1')));
	A_MV_1._sDescription	:= 	fcUtfToAscii(Standard.CONCAT(	OBJ_NAME_DESCRIPTION,	fcGetBcText(	GVL_BACNET.fbBacNetParameter.metGetTextListName(enTypeOfBacNetFunktionIn := enTypeOfBacNetFunktion.Type_Anlagenschalter,	enTypeOfBacNetTextListIn := enTypeOfBacNetTextList.DESCRIPTION	),	'A_MV_1')));
	(* Create Id from Base Id and Object Nr (Last nummber of Name *)	
	A_MV_1.Create(diInstance := TO_DINT(Standard.CONCAT(TO_STRING(dwOBJ_ID_BASE),'1')));
	(* Check if Created *)
	IF A_MV_1.xIsCreated THEN
		(* Set Group *)
		A_MV_1.setPropertyGroup(WagoTypesBacNet.eBACnetPropertyIdentifier.PROP_PRESENT_VALUE						,WagoTypesBacNet.eBACnetPropertyUpdateGroup.GROUP_CYCLIC);
		A_MV_1.setPropertyGroup(WagoTypesBacNet.eBACnetPropertyIdentifier.PROP_PRIORITY_ARRAY						,WagoTypesBacNet.eBACnetPropertyUpdateGroup.GROUP_CYCLIC);
		A_MV_1.setPropertyGroup(WagoTypesBacNet.eBACnetPropertyIdentifier.PROP_ELAPSED_ACTIVE_TIME					,WagoTypesBacNet.eBACnetPropertyUpdateGroup.GROUP_CYCLIC);
		A_MV_1.setPropertyGroup(WagoTypesBacNet.eBACnetPropertyIdentifier.PROP_DESCRIPTION							,WagoTypesBacNet.eBACnetPropertyUpdateGroup.GROUP_CYCLIC);
		A_MV_1.setPropertyGroup(WagoTypesBacNet.eBACnetPropertyIdentifier.PROP_EVENT_MESSAGE_TEXTS_CONFIG			,WagoTypesBacNet.eBACnetPropertyUpdateGroup.GROUP_CYCLIC);
		
		(* Set Description to Overwrite retain*)
		A_MV_1.sDescription	:= A_MV_1._sDescription;
		(* Ziel												UTF8->ASCII		BacNet Text		Textlistname									BacNet Funktion																BacNet Textlist type												TextId		*)
		A_MV_1.IEventMessageTextsConfig.sToOffNormal	:=	fcUtfToAscii(	fcGetBcText(	GVL_BACNET.fbBacNetParameter.metGetTextListName(enTypeOfBacNetFunktionIn := enTypeOfBacNetFunktion.Type_Anlagenschalter,	enTypeOfBacNetTextListIn := enTypeOfBacNetTextList.EVENTMESSAGE	),	'A_MV_1_ToOffNormal'	));		
		A_MV_1.IEventMessageTextsConfig.sToFault		:=	fcUtfToAscii(	fcGetBcText(	GVL_BACNET.fbBacNetParameter.metGetTextListName(enTypeOfBacNetFunktionIn := enTypeOfBacNetFunktion.Type_Anlagenschalter,	enTypeOfBacNetTextListIn := enTypeOfBacNetTextList.EVENTMESSAGE	),	'A_MV_1_ToFault'		));		
		A_MV_1.IEventMessageTextsConfig.sToNormal		:=	fcUtfToAscii(	fcGetBcText(	GVL_BACNET.fbBacNetParameter.metGetTextListName(enTypeOfBacNetFunktionIn := enTypeOfBacNetFunktion.Type_Anlagenschalter,	enTypeOfBacNetTextListIn := enTypeOfBacNetTextList.EVENTMESSAGE	),	'A_MV_1_ToNormal'		));		
		(* State Text *)
		A_MV_1.udiNumberOfStates						:= 	2;
		(* Ziel												UTF8->ASCII		BacNet Text		Textlistname									BacNet Funktion																BacNet Textlist type												TextId		*)	
		A_MV_1.setStateText(uiIndex	:= 1,	sStateText	:= 	fcUtfToAscii(	fcGetBcText(	GVL_BACNET.fbBacNetParameter.metGetTextListName(enTypeOfBacNetFunktionIn := enTypeOfBacNetFunktion.Type_Anlagenschalter,	enTypeOfBacNetTextListIn := enTypeOfBacNetTextList.PRESENTVALUE	),	'A_MV_1_ST_1'			)));
		A_MV_1.setStateText(uiIndex	:= 2,	sStateText	:= 	fcUtfToAscii(	fcGetBcText(	GVL_BACNET.fbBacNetParameter.metGetTextListName(enTypeOfBacNetFunktionIn := enTypeOfBacNetFunktion.Type_Anlagenschalter,	enTypeOfBacNetTextListIn := enTypeOfBacNetTextList.PRESENTVALUE	),	'A_MV_1_ST_2'			)));

	ELSE
		A_MV_1.Delete();
	END_IF;
	(* Get Status *)
	metCreate_A_MV_1 := A_MV_1.xIsCreated;	
END_IF;
END_METHOD

METHOD metCreate_B_MI_1 : BOOL
(* B_MI_1*)
IF NOT B_MI_1.xIsCreated THEN
	(* Ziel						UTF8->ASCII						OBJ_NAME_BASE			BacNet Text		Textlistname									BacNet Funktion																BacNet Textlist type												TextId		*)
	B_MI_1._sObjectName		:=	fcUtfToAscii(Standard.CONCAT(	OBJ_NAME_BASE		,	fcGetBcText(	GVL_BACNET.fbBacNetParameter.metGetTextListName(enTypeOfBacNetFunktionIn := enTypeOfBacNetFunktion.Type_Anlagenschalter,	enTypeOfBacNetTextListIn := enTypeOfBacNetTextList.ENDING		),	'B_MI_1')));
	B_MI_1._sDescription	:= 	fcUtfToAscii(Standard.CONCAT(	OBJ_NAME_DESCRIPTION,	fcGetBcText(	GVL_BACNET.fbBacNetParameter.metGetTextListName(enTypeOfBacNetFunktionIn := enTypeOfBacNetFunktion.Type_Anlagenschalter,	enTypeOfBacNetTextListIn := enTypeOfBacNetTextList.DESCRIPTION	),	'B_MI_1')));
	(* Create Id from Base Id and Object Nr (Last nummber of Name *)	
	B_MI_1.Create(diInstance := TO_DINT(Standard.CONCAT(TO_STRING(dwOBJ_ID_BASE),'1')));
	(* Check if Created *)
	IF B_MI_1.xIsCreated THEN
		(* Set Group *)
		B_MI_1.setPropertyGroup(WagoTypesBacNet.eBACnetPropertyIdentifier.PROP_PRESENT_VALUE						,WagoTypesBacNet.eBACnetPropertyUpdateGroup.GROUP_CYCLIC);
		B_MI_1.setPropertyGroup(WagoTypesBacNet.eBACnetPropertyIdentifier.PROP_PRIORITY_ARRAY						,WagoTypesBacNet.eBACnetPropertyUpdateGroup.GROUP_CYCLIC);
		B_MI_1.setPropertyGroup(WagoTypesBacNet.eBACnetPropertyIdentifier.PROP_ELAPSED_ACTIVE_TIME					,WagoTypesBacNet.eBACnetPropertyUpdateGroup.GROUP_CYCLIC);
		B_MI_1.setPropertyGroup(WagoTypesBacNet.eBACnetPropertyIdentifier.PROP_DESCRIPTION							,WagoTypesBacNet.eBACnetPropertyUpdateGroup.GROUP_CYCLIC);
		B_MI_1.setPropertyGroup(WagoTypesBacNet.eBACnetPropertyIdentifier.PROP_EVENT_MESSAGE_TEXTS_CONFIG			,WagoTypesBacNet.eBACnetPropertyUpdateGroup.GROUP_CYCLIC);
		
		(* Set Description to Overwrite retain*)
		B_MI_1.sDescription	:= B_MI_1._sDescription;
		(* Ziel												UTF8->ASCII		BacNet Text		Textlistname									BacNet Funktion																BacNet Textlist type												TextId		*)
		B_MI_1.IEventMessageTextsConfig.sToOffNormal	:=	fcUtfToAscii(	fcGetBcText(	GVL_BACNET.fbBacNetParameter.metGetTextListName(enTypeOfBacNetFunktionIn := enTypeOfBacNetFunktion.Type_Anlagenschalter,	enTypeOfBacNetTextListIn := enTypeOfBacNetTextList.EVENTMESSAGE	),	'B_MI_1_ToOffNormal'	));		
		B_MI_1.IEventMessageTextsConfig.sToFault		:=	fcUtfToAscii(	fcGetBcText(	GVL_BACNET.fbBacNetParameter.metGetTextListName(enTypeOfBacNetFunktionIn := enTypeOfBacNetFunktion.Type_Anlagenschalter,	enTypeOfBacNetTextListIn := enTypeOfBacNetTextList.EVENTMESSAGE	),	'B_MI_1_ToFault'		));		
		B_MI_1.IEventMessageTextsConfig.sToNormal		:=	fcUtfToAscii(	fcGetBcText(	GVL_BACNET.fbBacNetParameter.metGetTextListName(enTypeOfBacNetFunktionIn := enTypeOfBacNetFunktion.Type_Anlagenschalter,	enTypeOfBacNetTextListIn := enTypeOfBacNetTextList.EVENTMESSAGE	),	'B_MI_1_ToNormal'		));		
		(* State Text *)
		B_MI_1.udiNumberOfStates						:= 	3;
		(* Ziel												UTF8->ASCII		BacNet Text		Textlistname									BacNet Funktion																BacNet Textlist type												TextId		*)	
		B_MI_1.setStateText(uiIndex	:= 1,	sStateText	:= 	fcUtfToAscii(	fcGetBcText(	GVL_BACNET.fbBacNetParameter.metGetTextListName(enTypeOfBacNetFunktionIn := enTypeOfBacNetFunktion.Type_Anlagenschalter,	enTypeOfBacNetTextListIn := enTypeOfBacNetTextList.PRESENTVALUE	),	'B_MI_1_ST_1'			)));
		B_MI_1.setStateText(uiIndex	:= 2,	sStateText	:= 	fcUtfToAscii(	fcGetBcText(	GVL_BACNET.fbBacNetParameter.metGetTextListName(enTypeOfBacNetFunktionIn := enTypeOfBacNetFunktion.Type_Anlagenschalter,	enTypeOfBacNetTextListIn := enTypeOfBacNetTextList.PRESENTVALUE	),	'B_MI_1_ST_2'			)));
		B_MI_1.setStateText(uiIndex	:= 3,	sStateText	:= 	fcUtfToAscii(	fcGetBcText(	GVL_BACNET.fbBacNetParameter.metGetTextListName(enTypeOfBacNetFunktionIn := enTypeOfBacNetFunktion.Type_Anlagenschalter,	enTypeOfBacNetTextListIn := enTypeOfBacNetTextList.PRESENTVALUE	),	'B_MI_1_ST_3'			)));

	ELSE
		B_MI_1.Delete();
	END_IF;
	(* Get Status *)
	metCreate_B_MI_1 := B_MI_1.xIsCreated;	
END_IF;
END_METHOD

METHOD metCreate_C_BV_1 : BOOL
(* C_BV_1*)
IF NOT C_BV_1.xIsCreated THEN
	(* Ziel						UTF8->ASCII						OBJ_NAME_BASE			BacNet Text		Textlistname									BacNet Funktion																BacNet Textlist type												TextId		*)
	C_BV_1._sObjectName		:=	fcUtfToAscii(Standard.CONCAT(	OBJ_NAME_BASE		,	fcGetBcText(	GVL_BACNET.fbBacNetParameter.metGetTextListName(enTypeOfBacNetFunktionIn := enTypeOfBacNetFunktion.Type_Anlagenschalter,	enTypeOfBacNetTextListIn := enTypeOfBacNetTextList.ENDING		),	'C_BV_1')));
	C_BV_1._sDescription	:= 	fcUtfToAscii(Standard.CONCAT(	OBJ_NAME_DESCRIPTION,	fcGetBcText(	GVL_BACNET.fbBacNetParameter.metGetTextListName(enTypeOfBacNetFunktionIn := enTypeOfBacNetFunktion.Type_Anlagenschalter,	enTypeOfBacNetTextListIn := enTypeOfBacNetTextList.DESCRIPTION	),	'C_BV_1')));
	(* Create Id from Base Id and Object Nr (Last nummber of Name *)	
	C_BV_1.Create(diInstance := TO_DINT(Standard.CONCAT(TO_STRING(dwOBJ_ID_BASE),'1')));
	(* Check if Created *)
	IF C_BV_1.xIsCreated THEN
		(* Set Group *)
		C_BV_1.setPropertyGroup(WagoTypesBacNet.eBACnetPropertyIdentifier.PROP_PRESENT_VALUE						,WagoTypesBacNet.eBACnetPropertyUpdateGroup.GROUP_CYCLIC);
		C_BV_1.setPropertyGroup(WagoTypesBacNet.eBACnetPropertyIdentifier.PROP_PRIORITY_ARRAY						,WagoTypesBacNet.eBACnetPropertyUpdateGroup.GROUP_CYCLIC);
		C_BV_1.setPropertyGroup(WagoTypesBacNet.eBACnetPropertyIdentifier.PROP_ELAPSED_ACTIVE_TIME					,WagoTypesBacNet.eBACnetPropertyUpdateGroup.GROUP_CYCLIC);
		C_BV_1.setPropertyGroup(WagoTypesBacNet.eBACnetPropertyIdentifier.PROP_DESCRIPTION							,WagoTypesBacNet.eBACnetPropertyUpdateGroup.GROUP_CYCLIC);
		C_BV_1.setPropertyGroup(WagoTypesBacNet.eBACnetPropertyIdentifier.PROP_EVENT_MESSAGE_TEXTS_CONFIG			,WagoTypesBacNet.eBACnetPropertyUpdateGroup.GROUP_CYCLIC);
		
		(* Set Description to Overwrite retain*)
		C_BV_1.sDescription	:= C_BV_1._sDescription;
		(* Ziel												UTF8->ASCII		BacNet Text		Textlistname									BacNet Funktion																BacNet Textlist type												TextId		*)
		C_BV_1.IEventMessageTextsConfig.sToOffNormal	:=	fcUtfToAscii(	fcGetBcText(	GVL_BACNET.fbBacNetParameter.metGetTextListName(enTypeOfBacNetFunktionIn := enTypeOfBacNetFunktion.Type_Anlagenschalter,	enTypeOfBacNetTextListIn := enTypeOfBacNetTextList.EVENTMESSAGE	),	'C_BV_1_ToOffNormal'	));		
		C_BV_1.IEventMessageTextsConfig.sToFault		:=	fcUtfToAscii(	fcGetBcText(	GVL_BACNET.fbBacNetParameter.metGetTextListName(enTypeOfBacNetFunktionIn := enTypeOfBacNetFunktion.Type_Anlagenschalter,	enTypeOfBacNetTextListIn := enTypeOfBacNetTextList.EVENTMESSAGE	),	'C_BV_1_ToFault'		));		
		C_BV_1.IEventMessageTextsConfig.sToNormal		:=	fcUtfToAscii(	fcGetBcText(	GVL_BACNET.fbBacNetParameter.metGetTextListName(enTypeOfBacNetFunktionIn := enTypeOfBacNetFunktion.Type_Anlagenschalter,	enTypeOfBacNetTextListIn := enTypeOfBacNetTextList.EVENTMESSAGE	),	'C_BV_1_ToNormal'		));		
		(* Ziel												UTF8->ASCII		BacNet Text		Textlistname									BacNet Funktion																BacNet Textlist type												TextId		*)	
		C_BV_1.sActiveText								:= 	fcUtfToAscii(	fcGetBcText(	GVL_BACNET.fbBacNetParameter.metGetTextListName(enTypeOfBacNetFunktionIn := enTypeOfBacNetFunktion.Type_Anlagenschalter,	enTypeOfBacNetTextListIn := enTypeOfBacNetTextList.PRESENTVALUE	),	'C_BV_1_ST_ACTIVE'		));
		C_BV_1.sInactiveText							:= 	fcUtfToAscii(	fcGetBcText(	GVL_BACNET.fbBacNetParameter.metGetTextListName(enTypeOfBacNetFunktionIn := enTypeOfBacNetFunktion.Type_Anlagenschalter,	enTypeOfBacNetTextListIn := enTypeOfBacNetTextList.PRESENTVALUE	),	'C_BV_1_ST_INACTIVE'	));	
		(* Ziel												Convert			BacNet Text		Textlistname									BacNet Funktion																BacNet Textlist type												TextId		*)	
		C_BV_1.udiNotificationClass						:= 	TO_UDINT	(	fcGetBcText(	GVL_BACNET.fbBacNetParameter.metGetTextListName(enTypeOfBacNetFunktionIn := enTypeOfBacNetFunktion.Type_Anlagenschalter,	enTypeOfBacNetTextListIn := enTypeOfBacNetTextList.NC			),	'C_BV_1_NC'	));	
		C_BV_1.eNotifyType								:= 	WagoTypesBACnet.eBACnetNotifyType.NOTIFY_TYPE_EVENT;
		C_BV_1.xAlarmValue								:= 	TO_BOOL		(	fcGetBcText(	GVL_BACNET.fbBacNetParameter.metGetTextListName(enTypeOfBacNetFunktionIn := enTypeOfBacNetFunktion.Type_Anlagenschalter,	enTypeOfBacNetTextListIn := enTypeOfBacNetTextList.NC			),	'C_BV_1_ALV'	));			

	ELSE
		C_BV_1.Delete();
	END_IF;
	(* Get Status *)
	metCreate_C_BV_1 := C_BV_1.xIsCreated;	
END_IF;
END_METHOD

METHOD metCreate_D_SC_1 : BOOL
(* D_SC_1*)
IF NOT D_SC_1.xIsCreated THEN
	(* Ziel						UTF8->ASCII						OBJ_NAME_BASE			BacNet Text		Textlistname									BacNet Funktion																BacNet Textlist type												TextId		*)
	D_SC_1._sObjectName		:=	fcUtfToAscii(Standard.CONCAT(	OBJ_NAME_BASE		,	fcGetBcText(	GVL_BACNET.fbBacNetParameter.metGetTextListName(enTypeOfBacNetFunktionIn := enTypeOfBacNetFunktion.Type_Anlagenschalter,	enTypeOfBacNetTextListIn := enTypeOfBacNetTextList.ENDING		),	'D_SC_1')));
	D_SC_1._sDescription	:= 	fcUtfToAscii(Standard.CONCAT(	OBJ_NAME_DESCRIPTION,	fcGetBcText(	GVL_BACNET.fbBacNetParameter.metGetTextListName(enTypeOfBacNetFunktionIn := enTypeOfBacNetFunktion.Type_Anlagenschalter,	enTypeOfBacNetTextListIn := enTypeOfBacNetTextList.DESCRIPTION	),	'D_SC_1')));
	(* Create Id from Base Id and Object Nr (Last nummber of Name *)	
	D_SC_1.Create(diInstance := TO_DINT(Standard.CONCAT(TO_STRING(dwOBJ_ID_BASE),'1')));
	(* Check if Created *)
	IF D_SC_1.xIsCreated THEN
		(* Set Group *)
		D_SC_1.setPropertyGroup(WagoTypesBacNet.eBACnetPropertyIdentifier.PROP_PRESENT_VALUE						,WagoTypesBacNet.eBACnetPropertyUpdateGroup.GROUP_CYCLIC);
		D_SC_1.setPropertyGroup(WagoTypesBacNet.eBACnetPropertyIdentifier.PROP_PRIORITY_ARRAY						,WagoTypesBacNet.eBACnetPropertyUpdateGroup.GROUP_CYCLIC);
		D_SC_1.setPropertyGroup(WagoTypesBacNet.eBACnetPropertyIdentifier.PROP_ELAPSED_ACTIVE_TIME					,WagoTypesBacNet.eBACnetPropertyUpdateGroup.GROUP_CYCLIC);
		D_SC_1.setPropertyGroup(WagoTypesBacNet.eBACnetPropertyIdentifier.PROP_DESCRIPTION							,WagoTypesBacNet.eBACnetPropertyUpdateGroup.GROUP_CYCLIC);
		D_SC_1.setPropertyGroup(WagoTypesBacNet.eBACnetPropertyIdentifier.PROP_EVENT_MESSAGE_TEXTS_CONFIG			,WagoTypesBacNet.eBACnetPropertyUpdateGroup.GROUP_CYCLIC);
		
		(* Set Description to Overwrite retain*)
		D_SC_1.sDescription	:= D_SC_1._sDescription;
		(* Ziel												UTF8->ASCII		BacNet Text		Textlistname									BacNet Funktion																BacNet Textlist type												TextId		*)
		D_SC_1.IEventMessageTextsConfig.sToOffNormal	:=	fcUtfToAscii(	fcGetBcText(	GVL_BACNET.fbBacNetParameter.metGetTextListName(enTypeOfBacNetFunktionIn := enTypeOfBacNetFunktion.Type_Anlagenschalter,	enTypeOfBacNetTextListIn := enTypeOfBacNetTextList.EVENTMESSAGE	),	'D_SC_1_ToOffNormal'	));		
		D_SC_1.IEventMessageTextsConfig.sToFault		:=	fcUtfToAscii(	fcGetBcText(	GVL_BACNET.fbBacNetParameter.metGetTextListName(enTypeOfBacNetFunktionIn := enTypeOfBacNetFunktion.Type_Anlagenschalter,	enTypeOfBacNetTextListIn := enTypeOfBacNetTextList.EVENTMESSAGE	),	'D_SC_1_ToFault'		));		
		D_SC_1.IEventMessageTextsConfig.sToNormal		:=	fcUtfToAscii(	fcGetBcText(	GVL_BACNET.fbBacNetParameter.metGetTextListName(enTypeOfBacNetFunktionIn := enTypeOfBacNetFunktion.Type_Anlagenschalter,	enTypeOfBacNetTextListIn := enTypeOfBacNetTextList.EVENTMESSAGE	),	'D_SC_1_ToNormal'		));		

	ELSE
		D_SC_1.Delete();
	END_IF;
	(* Get Status *)
	metCreate_D_SC_1 := D_SC_1.xIsCreated;	
END_IF;
END_METHOD

METHOD metCREATE_KBOB_2017_V1 : BOOL;
VAR_INPUT
END_VAR
VAR
	oStatus		:	WagoSysErrorBase.FbResult;
	usiErrors	:	USINT;
END_VAR
(* Resett *)
usiErrors := 0;	

(* Create Objeccts *)
CASE usiCreateCase OF
	1:
		usiErrors := usiErrors + TO_USINT(NOT metCreate_A_MV_1());
	2:
		usiErrors := usiErrors + TO_USINT(NOT metCreate_B_MI_1());
	3:
		usiErrors := usiErrors + TO_USINT(NOT metCreate_C_BV_1());
	4:
		usiErrors := usiErrors + TO_USINT(NOT metCreate_D_SC_1());
	0: 
		usiCreateCase := 1;
ELSE
	usiCreateCase := 0;
END_CASE;

(* STRUCT VIEW *)
metCREATE_STRUCTVIEW_KBOB_2017_V1();

(* OK = 0*)
metCREATE_KBOB_2017_V1 := NOT TO_BOOL(usiErrors);
END_METHOD

METHOD metCREATE_STRUCTVIEW_KBOB_2017_V1 : BOOL
VAR_INPUT
END_VAR
CASE usiCreateCase OF
	1:
		fcXMLStructuredView(THIS^,A_MV_1.IObjectIdentifier);
	2:
		fcXMLStructuredView(THIS^,B_MI_1.IObjectIdentifier);
	3:
		fcXMLStructuredView(THIS^,C_BV_1.IObjectIdentifier);
	4:
		fcXMLStructuredView(THIS^,D_SC_1.IObjectIdentifier);
		fcXMLAddStructuredViewToDevice(THIS^);	
	0: 
		usiCreateCase := 1;
ELSE
	usiCreateCase := 0;
END_CASE
END_METHOD

METHOD metCREATE_KBOB_2021_V2 : BOOL;
VAR_INPUT
END_VAR
VAR
	oStatus		:	WagoSysErrorBase.FbResult;
	usiErrors	:	USINT;
END_VAR
(* Resett *)
usiErrors := 0;	

(* Create Objeccts *)
CASE usiCreateCase OF
	1:
		usiErrors := usiErrors + TO_USINT(NOT metCreate_A_MV_1());
	2:
		usiErrors := usiErrors + TO_USINT(NOT metCreate_B_MI_1());
	3:
		usiErrors := usiErrors + TO_USINT(NOT metCreate_C_BV_1());
	4:
		usiErrors := usiErrors + TO_USINT(NOT metCreate_D_SC_1());
	0: 
		usiCreateCase := 1;
ELSE
	usiCreateCase := 0;
END_CASE;

(* STRUCT VIEW *)
metCREATE_STRUCTVIEW_KBOB_2021_V2();

(* OK = 0*)
metCREATE_KBOB_2021_V2 := NOT TO_BOOL(usiErrors);
END_METHOD

METHOD metCREATE_STRUCTVIEW_KBOB_2021_V2 : BOOL
VAR_INPUT
END_VAR
CASE usiCreateCase OF
	1:
		fcXMLStructuredView(THIS^,A_MV_1.IObjectIdentifier);
	2:
		fcXMLStructuredView(THIS^,B_MI_1.IObjectIdentifier);
	3:
		fcXMLStructuredView(THIS^,C_BV_1.IObjectIdentifier);
	4:
		fcXMLStructuredView(THIS^,D_SC_1.IObjectIdentifier);
		fcXMLAddStructuredViewToDevice(THIS^);	
	0: 
		usiCreateCase := 1;
ELSE
	usiCreateCase := 0;
END_CASE
END_METHOD

METHOD metDELETE : BOOL
VAR_INPUT
END_VAR
VAR
	oStatus		:	WagoSysErrorBase.FbResult;
END_VAR
(* A_MV_1*)
IF A_MV_1.xIsCreated THEN
	A_MV_1.Delete(oStatus=>oStatus);
END_IF;	
(* B_MI_1 *)
IF B_MI_1.xIsCreated THEN
		B_MI_1.Delete(oStatus=>oStatus);
END_IF;	
(* C_BV_1 *)
IF C_BV_1.xIsCreated THEN
	C_BV_1.Delete(oStatus=>oStatus);
END_IF;
(* D_SC_1 *)
IF D_SC_1.xIsCreated THEN
	D_SC_1.Delete(oStatus=>oStatus);	
END_IF;
(* Delete Struct View *)
IF GVL_BACNET.fbBacNetParameter.proDestroyBacNetOverrideXmlNode THEN
	fcXMLDeleteOverrideNode(fcBacNetIdToIdWitType(TO_DINT(CONCAT(TO_STRING(OBJ_ID_BASE),'1')),WagoTypesBacNet.eBACnetObjectType.BACnet_structured_view));
	fcXMLDeleteStructuredViewFromDevice(fcBacNetIdToIdWitType(TO_DINT(CONCAT(TO_STRING(OBJ_ID_BASE),'1')),WagoTypesBacNet.eBACnetObjectType.BACnet_structured_view));
END_IF;
metDELETE := 	A_MV_1.xIsCreated OR
				B_MI_1.xIsCreated OR
				C_BV_1.xIsCreated OR
				D_SC_1.xIsCreated ;
(* Reset Create Case *)
usiCreateCase := 1;
END_METHOD

METHOD metCYCLIC_KBOB_2017_V1
VAR_INPUT
END_VAR
(* A_MV_1 *)
IF A_MV_1.udiNumberOfStates <> 2 THEN
	A_MV_1.udiNumberOfStates := 2;
END_IF;	
(* Auto *)
IF xAutoIn THEN	
	IF A_MV_1.IPriorityArray.aLevel[16].xNull <> xAutoIn THEN
		A_MV_1.IPriorityArray.SetPriority(16,0,TRUE);
	END_IF;
	(* Check if in Service *)
	IF NOT D_SC_1.xOutOfService THEN
		(* Check if not Null *)
		IF D_SC_1.IPresentValue.eDataType <> WagoTypesBACnet.eBACnetDataType.BACNET_TYPE_NULL THEN
			(* Check if right Data Type *)
			IF D_SC_1.IPresentValue.eDataType = WagoTypesBACnet.eBACnetDataType.BACNET_TYPE_UNSIGNED THEN 
				(* Set Scheduler state in Prio 14 *)
				IF A_MV_1.IPriorityArray.aLevel[14].xNull OR A_MV_1.IPriorityArray.aLevel[14].udiValue <> D_SC_1.IPresentValue.IUNSIGNED.udiValue THEN
					A_MV_1.IPriorityArray.SetPriority(14,D_SC_1.IPresentValue.IUNSIGNED.udiValue,FALSE);
				END_IF;
			END_IF;
		ELSE
			(* Set Prio 14 NULL *)
			IF NOT A_MV_1.IPriorityArray.aLevel[14].xNull THEN
				A_MV_1.IPriorityArray.SetPriority(14,1,TRUE);
			END_IF;		
		END_IF;
	ELSE
		(* Set Prio 14 NULL *)
		IF NOT A_MV_1.IPriorityArray.aLevel[14].xNull THEN
			A_MV_1.IPriorityArray.SetPriority(14,1,TRUE);
		END_IF;			
	END_IF;
(* Hand Aus *)
ELSIF xHandOffIn THEN
	(* Get State of A_MV_1 at level 16 and set new State if necesseray *)
	IF A_MV_1.IPriorityArray.aLevel[16].xNull OR A_MV_1.IPriorityArray.aLevel[16].udiValue <> 1 THEN
		A_MV_1.IPriorityArray.SetPriority(16,1,FALSE);
	END_IF;
(* Hand Ein *)		
ELSIF xHandOnIn THEN
	(* Get State of A_MV_1 at level 16 and set new State if necesseray *)
	IF A_MV_1.IPriorityArray.aLevel[16].xNull OR A_MV_1.IPriorityArray.aLevel[16].udiValue <> 2  THEN
		A_MV_1.IPriorityArray.SetPriority(16,2,FALSE);
	END_IF;		
ELSE
	(* Get State of A_MV_1 at level 16 and set new State if necesseray *)
	IF A_MV_1.IPriorityArray.aLevel[16].xNull OR A_MV_1.IPriorityArray.aLevel[16].udiValue <> 1  THEN
		A_MV_1.IPriorityArray.SetPriority(16,1,FALSE);
	END_IF;	
END_IF;

(* B_MI_1 *)
IF B_MI_1.udiNumberOfStates <> 3 THEN
	B_MI_1.udiNumberOfStates := 3;
END_IF;

(* Set Local Auto *)
IF xAutoIn THEN
	IF B_MI_1.udiPresentValue <> 1 THEN
		B_MI_1.udiPresentValue := 1;		(* Auto Lokal *)			
	END_IF;
	IF NOT A_MV_1.IPriorityArray.aLevel[7].xNull THEN
		A_MV_1.IPriorityArray.SetPriority(7,0,TRUE);
	END_IF;
(* Set Local Hand Off *)
ELSIF xHandOffIn THEN
	IF B_MI_1.udiPresentValue <> 2 THEN
		B_MI_1.udiPresentValue := 2;		(* Aus Lokal *)
	END_IF;
	IF A_MV_1.IPriorityArray.aLevel[7].xNull OR A_MV_1.IPriorityArray.aLevel[7].udiValue <> 1 THEN
		A_MV_1.IPriorityArray.SetPriority(7,1,FALSE);	
	END_IF
(* Set Local Hadn On *)
ELSIF xHandOnIn THEN
	IF B_MI_1.udiPresentValue <> 3 THEN
		B_MI_1.udiPresentValue := 3;		(* Ein Lokal *)
	END_IF;
	IF A_MV_1.IPriorityArray.aLevel[7].xNull OR A_MV_1.IPriorityArray.aLevel[7].udiValue <> 2 THEN
		A_MV_1.IPriorityArray.SetPriority(7,2,FALSE);	
	END_IF		
END_IF;

(* C_BV_1 *)
IF NOT A_MV_1.IPriorityArray.aLevel[7].xNull OR NOT A_MV_1.IPriorityArray.aLevel[8].xNull THEN
	IF C_BV_1.xPresentValue = FALSE	THEN
		(* Notification Hand *)
		C_BV_1.xPresentValue := TRUE;
	END_IF;
ELSE
	IF C_BV_1.xPresentValue = TRUE THEN
		(* Notification Auto *)
		C_BV_1.xPresentValue := FALSE;
	END_IF;
END_IF;

(* State Out *)
IF C_BV_1.xPresentValue THEN
	xOffOut	 := A_MV_1.udiPresentValue = 1;
	xOnOut	 := A_MV_1.udiPresentValue = 2;	
	xAutoOut := FALSE;
	xHandOut := TRUE;
ELSE
	xAutoOut := TRUE;
	xHandOut := FALSE;
	xOnOut	 := A_MV_1.udiPresentValue = 2;	
	xOffOut	 := NOT xOnOut;	
END_IF;
END_METHOD

METHOD metCYCLIC_KBOB_2021_V2
VAR_INPUT
END_VAR
(* A_MV_1 *)
IF A_MV_1.udiNumberOfStates <> 2 THEN
	A_MV_1.udiNumberOfStates := 2;
END_IF;	
(* Auto *)
IF xAutoIn THEN	
	IF A_MV_1.IPriorityArray.aLevel[16].xNull <> xAutoIn THEN
		A_MV_1.IPriorityArray.SetPriority(16,0,TRUE);
	END_IF;
	(* Check if in Service *)
	IF NOT D_SC_1.xOutOfService THEN
		(* Check if not Null *)
		IF D_SC_1.IPresentValue.eDataType <> WagoTypesBACnet.eBACnetDataType.BACNET_TYPE_NULL THEN
			(* Check if right Data Type *)
			IF D_SC_1.IPresentValue.eDataType = WagoTypesBACnet.eBACnetDataType.BACNET_TYPE_UNSIGNED THEN 
				(* Set Scheduler state in Prio 14 *)
				IF A_MV_1.IPriorityArray.aLevel[14].xNull OR A_MV_1.IPriorityArray.aLevel[14].udiValue <> D_SC_1.IPresentValue.IUNSIGNED.udiValue THEN
					A_MV_1.IPriorityArray.SetPriority(14,D_SC_1.IPresentValue.IUNSIGNED.udiValue,FALSE);
				END_IF;
			END_IF;
		ELSE
			(* Set Prio 14 NULL *)
			IF NOT A_MV_1.IPriorityArray.aLevel[14].xNull THEN
				A_MV_1.IPriorityArray.SetPriority(14,1,TRUE);
			END_IF;		
		END_IF;
	ELSE
		(* Set Prio 14 NULL *)
		IF NOT A_MV_1.IPriorityArray.aLevel[14].xNull THEN
			A_MV_1.IPriorityArray.SetPriority(14,1,TRUE);
		END_IF;			
	END_IF;
(* Hand Aus *)
ELSIF xHandOffIn THEN
	(* Get State of A_MV_1 at level 16 and set new State if necesseray *)
	IF A_MV_1.IPriorityArray.aLevel[16].xNull OR A_MV_1.IPriorityArray.aLevel[16].udiValue <> 1 THEN
		A_MV_1.IPriorityArray.SetPriority(16,1,FALSE);
	END_IF;
(* Hand Ein *)		
ELSIF xHandOnIn THEN
	(* Get State of A_MV_1 at level 16 and set new State if necesseray *)
	IF A_MV_1.IPriorityArray.aLevel[16].xNull OR A_MV_1.IPriorityArray.aLevel[16].udiValue <> 2  THEN
		A_MV_1.IPriorityArray.SetPriority(16,2,FALSE);
	END_IF;		
ELSE
	(* Get State of A_MV_1 at level 16 and set new State if necesseray *)
	IF A_MV_1.IPriorityArray.aLevel[16].xNull OR A_MV_1.IPriorityArray.aLevel[16].udiValue <> 1  THEN
		A_MV_1.IPriorityArray.SetPriority(16,1,FALSE);
	END_IF;	
END_IF;

(* B_MI_1 *)
IF B_MI_1.udiNumberOfStates <> 3 THEN
	B_MI_1.udiNumberOfStates := 3;
END_IF;

(* Set Local Auto *)
IF xAutoIn THEN
	IF B_MI_1.udiPresentValue <> 1 THEN
		B_MI_1.udiPresentValue := 1;		(* Auto Lokal *)			
	END_IF;
	IF NOT A_MV_1.IPriorityArray.aLevel[7].xNull THEN
		A_MV_1.IPriorityArray.SetPriority(7,0,TRUE);
	END_IF;
(* Set Local Hand Off *)
ELSIF xHandOffIn THEN
	IF B_MI_1.udiPresentValue <> 2 THEN
		B_MI_1.udiPresentValue := 2;		(* Aus Lokal *)
	END_IF;
	IF A_MV_1.IPriorityArray.aLevel[7].xNull OR A_MV_1.IPriorityArray.aLevel[7].udiValue <> 1 THEN
		A_MV_1.IPriorityArray.SetPriority(7,1,FALSE);	
	END_IF
(* Set Local Hadn On *)
ELSIF xHandOnIn THEN
	IF B_MI_1.udiPresentValue <> 3 THEN
		B_MI_1.udiPresentValue := 3;		(* Ein Lokal *)
	END_IF;
	IF A_MV_1.IPriorityArray.aLevel[7].xNull OR A_MV_1.IPriorityArray.aLevel[7].udiValue <> 2 THEN
		A_MV_1.IPriorityArray.SetPriority(7,2,FALSE);	
	END_IF		
END_IF;

(* C_BV_1 *)
IF NOT A_MV_1.IPriorityArray.aLevel[7].xNull OR NOT A_MV_1.IPriorityArray.aLevel[8].xNull THEN
	IF C_BV_1.xPresentValue = FALSE	THEN
		(* Notification Hand *)
		C_BV_1.xPresentValue := TRUE;
	END_IF;
ELSE
	IF C_BV_1.xPresentValue = TRUE THEN
		(* Notification Auto *)
		C_BV_1.xPresentValue := FALSE;
	END_IF;
END_IF;

(* State Out *)
IF C_BV_1.xPresentValue THEN
	xOffOut	 := A_MV_1.udiPresentValue = 1;
	xOnOut	 := A_MV_1.udiPresentValue = 2;	
	xAutoOut := FALSE;
	xHandOut := TRUE;
ELSE
	xAutoOut := TRUE;
	xHandOut := FALSE;
	xOnOut	 := A_MV_1.udiPresentValue = 2;	
	xOffOut	 := NOT xOnOut;	
END_IF;
END_METHOD

METHOD metCYCLIC_DESCRIPTION_FIX
VAR_INPUT
END_VAR
(* A_MV_1 *)
IF A_MV_1.xIsCreated THEN
	IF A_MV_1.sDescription <> A_MV_1._sDescription THEN
		A_MV_1.sDescription := A_MV_1._sDescription;
	END_IF;
END_IF;

(* B_MI_1 *)
IF B_MI_1.xIsCreated THEN
	IF B_MI_1.sDescription <> B_MI_1._sDescription THEN
		B_MI_1.sDescription := B_MI_1._sDescription;
	END_IF;
END_IF;

(* C_BV_1 *)
IF C_BV_1.xIsCreated THEN
	IF C_BV_1.sDescription <> C_BV_1._sDescription THEN
		C_BV_1.sDescription := C_BV_1._sDescription;
	END_IF;
END_IF;

(* D_SC_1 *)
IF D_SC_1.xIsCreated THEN
	IF D_SC_1.sDescription <> D_SC_1._sDescription THEN
		D_SC_1.sDescription := D_SC_1._sDescription;
	END_IF;
END_IF;
END_METHOD

END_FUNCTION_BLOCK

// 30 Program Organization Units/FCs/UTF8Fcs/fcAsciiToUtf
FUNCTION fcAsciiToUtf : STRING(255)
VAR_INPUT
	stIn	:	STRING(255);
END_VAR
VAR
	stFind	:	STRING(1);
	iSafety	:	INT;
	iPos	:	INT;
	iLen	:	INT;
END_VAR

IF GVL_BACNET.fbBacNetParameter.fbxAnsiCodiert.proValue THEN
	(* Ä *)
	IF Standard.LEN('Ä') <> 1 THEN	// Check if UTF 8 = 2 Byte or ASCII = 1 Byte
		iSafety := 0;
		stFind[0] := 196;	// ANSI Ä
		WHILE Standard.FIND(stIn,stFind) <> 0 AND iSafety < 255 DO	
			iPos 		:= Standard.FIND(stIn,stFind)-1;
			stIn 		:= Standard.DELETE(stIn,Standard.LEN(stFind),Standard.FIND(stIn,stFind));
			stIn		:= Standard.INSERT(stIn,'Ä',iPos);
			iSafety := iSafety + 1;
		END_WHILE;
	END_IF;
	IF Standard.LEN('ä') <> 1 THEN 	// Check if UTF 8 = 2 Byte or ASCII = 1 Byte
		iSafety := 0;
		stFind[0] := 228;	// ANSI ä
		WHILE Standard.FIND(stIn,'ä') <> 0 AND iSafety < 255 DO	
			iPos 		:= Standard.FIND(stIn,stFind)-1;
			stIn 		:= Standard.DELETE(stIn,Standard.LEN(stFind),Standard.FIND(stIn,stFind));
			stIn		:= Standard.INSERT(stIn,'ä',iPos);
			iSafety := iSafety + 1;
		END_WHILE;
	END_IF;
	(* Ö *)
	IF Standard.LEN('Ö') <> 1 THEN	// Check if UTF 8 = 2 Byte or ASCII = 1 Byte
		iSafety := 0;
		stFind[0] := 214;	// ANSI Ö
		WHILE Standard.FIND(stIn,'Ö') <> 0 AND iSafety < 255 DO	
			iPos 		:= Standard.FIND(stIn,stFind)-1;
			stIn 		:= Standard.DELETE(stIn,Standard.LEN(stFind),Standard.FIND(stIn,stFind));
			stIn		:= Standard.INSERT(stIn,'Ö',iPos);
			iSafety := iSafety + 1;
		END_WHILE;
	END_IF;
	IF Standard.LEN('ö') <> 1 THEN	// Check if UTF 8 = 2 Byte or ASCII = 1 Byte
		iSafety := 0;
		stFind[0] := 246;	// ANSI ö
		WHILE Standard.FIND(stIn,'ö') <> 0 AND iSafety < 255 DO	
			iPos 		:= Standard.FIND(stIn,stFind)-1;
			stIn 		:= Standard.DELETE(stIn,Standard.LEN(stFind),Standard.FIND(stIn,stFind));
			stIn		:= Standard.INSERT(stIn,'ö',iPos);
			iSafety := iSafety + 1;
		END_WHILE;
	END_IF;
	(* Ü *)
	IF Standard.LEN('Ü') <> 1 THEN	// Check if UTF 8 = 2 Byte or ASCII = 1 Byte
		iSafety := 0;
		stFind[0] := 220;	// ANSI Ü
		WHILE Standard.FIND(stIn,'Ü') <> 0 AND iSafety < 255 DO	
			iPos 		:= Standard.FIND(stIn,stFind)-1;
			stIn 		:= Standard.DELETE(stIn,Standard.LEN(stFind),Standard.FIND(stIn,stFind));
			stIn		:= Standard.INSERT(stIn,'Ü',iPos);
			iSafety := iSafety + 1;
		END_WHILE;
	END_IF;
	IF Standard.LEN('ü') <> 1 THEN	// Check if UTF 8 = 2 Byte or ASCII = 1 Byte
		iSafety := 0;
		stFind[0] := 252;	// ANSI ü
		WHILE Standard.FIND(stIn,'ü') <> 0 AND iSafety < 255 DO	
			iPos 		:= Standard.FIND(stIn,stFind)-1;
			stIn 		:= Standard.DELETE(stIn,Standard.LEN(stFind),Standard.FIND(stIn,stFind));
			stIn		:= Standard.INSERT(stIn,'ü',iPos);
			iSafety := iSafety + 1;
		END_WHILE;
	END_IF;
END_IF;
fcAsciiToUtf := stIn;

END_FUNCTION

// 30 Program Organization Units/FBs/BACNET_PARAMETER/FB_BACNET_PARAMETER
FUNCTION_BLOCK FB_BACNET_PARAMETER IMPLEMENTS ITF_BACNET_PARAMETER
VAR_INPUT
END_VAR
VAR_OUTPUT
END_VAR
VAR
	xInitDone					:	BOOL;
	xWarningParameter			:	BOOL;
	xPeresistenceOverride		:	BOOL;
	xCreate						:	BOOL;
	xDelete						:	BOOL;
	xDestroyBacNetOverrideNode	:	BOOL;
	xRebootRequired				:	BOOL;
	uiCountObj					:	UINT;
	uiCountCreatetObj			:	UINT;
	uiCountDeleteObj			:	UINT;
	TON_DELAY_START				:	Standard.TON;
	xUseExklTxtListOld			:	BOOL;
	xUseAksOld					:	BOOL;
	xReloadOnChange				:	BOOL;
	xDeleteLock					:	BOOL;
	fbConfigFile				:	CtaSysConfig.fbConfigFile;
	fbxEnableBacNet				:	CtaSysConfig.fbBOOL;
	fbxUseAKS					:	CtaSysConfig.fbBOOL;
	fbxUseExklTxtList			:	CtaSysConfig.fbBOOL;
	fbenBacNetKbobRev			:	CtaSysConfig.fbINT;
	fbdiDeviceId				:	CtaSysConfig.fbDINT;
	fbxAnsiCodiert				:	CtaSysConfig.fbBOOL;
	
	ITF_FIRST_OBJ				:	ITF_OBJ_ID_BASE	:= 0;
	ITF_NEXT_OBJ				:	ITF_OBJ_ID_BASE	:= 0;
	ITF_CREATE_OBJ				:	ITF_OBJ_ID_BASE	:= 0;
	ITF_TEMP_OBJ				:	ITF_OBJ_ID_BASE	:= 0;
	
	error						:	WagoSysBACnet.eErrorBACnet;	
END_VAR

(* Config *)			
CONFIG();
(* Delay *)
TON_DELAY_START(IN	:= NOT xReloadOnChange,
				PT  := T#20S);
IF NOT xPeresistenceOverride THEN
	fcXMLUpdateAttribute('/','wagoDevice','','','persistency','2','/home/user/bacnet/config/override.xml');
	fcBacNetIni();
	xPeresistenceOverride := TRUE;
END_IF
(* Enable BacNet *)
IF fbxEnableBacNet.proValue AND TON_DELAY_START.Q THEN
	xCreate := TRUE;
	xDelete := FALSE;
	xDestroyBacNetOverrideNode := FALSE;	
	IF uiCountCreatetObj < uiCountObj THEN
		(* iterate all connectet AT Function Blocks *)
		IF __QUERYINTERFACE(ITF_FIRST_OBJ,ITF_FIRST_OBJ) THEN
			IF __QUERYINTERFACE(ITF_CREATE_OBJ,ITF_CREATE_OBJ) THEN
				IF NOT ITF_CREATE_OBJ.proIsCreatet THEN
					ITF_CREATE_OBJ.proAllowCreate := TRUE;
				ELSE
					IF __QUERYINTERFACE(ITF_CREATE_OBJ,ITF_TEMP_OBJ) THEN
						ITF_CREATE_OBJ := ITF_TEMP_OBJ.proINextObj;
						uiCountCreatetObj := uiCountCreatetObj + 1;
					END_IF;
				END_IF;
			ELSE
				IF NOT ITF_FIRST_OBJ.proIsCreatet THEN
					ITF_FIRST_OBJ.proAllowCreate := TRUE;
				ELSE
					ITF_CREATE_OBJ := ITF_FIRST_OBJ.proINextObj;
					uiCountCreatetObj := uiCountCreatetObj + 1;
				END_IF;
			END_IF;
		END_IF;
	ELSE
		ITF_CREATE_OBJ	:= 0;
		ITF_TEMP_OBJ	:= 0;
	END_IF;		
	uiCountDeleteObj := 0;
ELSE
	IF xCreate THEN
		xCreate	:= FALSE;
		xDelete := TRUE;
		xDestroyBacNetOverrideNode := TRUE;
		ITF_CREATE_OBJ	:= 0;
		ITF_TEMP_OBJ	:= 0;			
		uiCountCreatetObj := 0;		
	END_IF;
END_IF

PROPERTY proCreate : Bool
GET
proCreate := xCreate;
END_GET
END_PROPERTY

PROPERTY proDelete : Bool
GET
proDelete := xDelete;
END_GET
END_PROPERTY

PROPERTY proUseAKS : BOOL
GET
proUseAKS := fbxUseAKS.xValue;
END_GET
END_PROPERTY

PROPERTY proInitDone : BOOL
GET
proInitDone := xInitDone;
END_GET
END_PROPERTY

ACTION CONFIG:
(* Config File *)
fbConfigFile();
fbxEnableBacNet		(_usiParaNr := 1,itfConfigFb := fbConfigFile);
fbxUseAKS			(_usiParaNr := 2,itfConfigFb := fbConfigFile);
fbxUseExklTxtList	(_usiParaNr := 3,itfConfigFb := fbConfigFile);
fbenBacNetKbobRev	(_usiParaNr := 4,itfConfigFb := fbConfigFile);
fbdiDeviceId		(_usiParaNr := 5,itfConfigFb := fbConfigFile,_MinInit := 0,_MaxInit := 4194302);
fbxAnsiCodiert	(_usiParaNr := 6,itfConfigFb := fbConfigFile,_WertInit := TRUE);
(* Check if Parameter Change *)
IF fbxEnableBacNet.proStateChanged 		OR 
	fbxUseExklTxtList.proStateChanged 	OR 
	fbxUseAKS.proStateChanged 			OR 
	fbenBacNetKbobRev.proStateChanged 	OR
	fbdiDeviceId.proStateChanged 		OR 
	fbxAnsiCodiert.proStateChanged		THEN
	xInitDone 					:= FALSE;
	xUseExklTxtListOld 			:= fbxUseExklTxtList.xValue; 
	xUseAksOld 					:= fbxUseAKS.xValue;
	xReloadOnChange				:= TRUE;
ELSE
	xInitDone	 		:= TRUE;
	xReloadOnChange		:= FALSE;
END_IF;
END_ACTION

METHOD metRequestDelete : BOOL
metRequestDelete := NOT xDeleteLock;
IF metRequestDelete THEN
	xDeleteLock := TRUE;
END_IF;
END_METHOD

